(* IEC 61131-3 sources: Mizera_Tube/Plc, 88 files *)

(* ---- Aspiraz.plc ---- *)
*******************************************************************************
*   ASPIRAZ.PLC
*   ESAutomotion
*   LASER machine
*******************************************************************************
#funcdec "SetVasca.plc"

VAR
#include "Cnc.inc"

EXHAUST_MNGT:           EXHAUST;    * Vasche di aspirazione
TimeOff:                DWORD;
TON_ASP:                TON;
TON_ASPI:               TON;
TOF_ASPI:               TOF;
TON_PROGRUN:            TON;
TOF_EXEAUTO:            TOF;
appoggio:               BOOL;
END_VAR

#include "Iol.inc"
#include "Aspiraz.inc"

VAR_IN_OUT
#include "mem.inc"
END_VAR
*******************************************************************************
* Gestione Aspirazione
*******************************************************************************
FUNCTION Aspiraz

*******************************************************************************
*   Richiesta da Pulsante Aspirazione ON\OFF
*******************************************************************************

CAL  TON_PROGRUN (IN:=PRGRUN_CN0,PT:=200)
CAL  TOF_EXEAUTO (IN:=ExeAuxMode,PT:=1000)

LD   Pls_ON_OFF_Aspiratore         ** (LsGui0.31)Pulsante ON\OFF accensione Aspiratore
OR   (
LD   Pls_AspAuto                   ** (rLsGui0.11) Pulsante Abilitazione Auto Aspiratore
AND  TON_PROGRUN.Q
ANDN TOF_EXEAUTO.Q
OR (
LD   ExeAuxMode                    ** (gPlc0.29)Esecuzione ausiliaria 1000.PGM
AND  exeaux_for_mancut               ** (LsPlc47.8) manual cut request
)
)
ANDN %PlcOp0.2                     ** DryRun
ST   appoggio

LD   %Cost_User9
MUL  1000
ST   TimeOff

CAL  TON_ASPI (IN:=appoggio,PT:=100)
CAL  TOF_ASPI (IN:=TON_ASPI.Q,PT:=TimeOff)

LD   TOF_ASPI.Q
ST   O_START_ASPIRATORE            ** Command START for Aspiration system
ST   AspOnOffLED                   ** (LsPlc11.17) LED Comando ON\OFF Aspiratore

LDN  O_START_ASPIRATORE            ** Command START for Aspiration system
ST   O_STOP_ASPIRATORE             ** Command STOP for Aspiration system

***************************************
*   EXHAUST FAN
***************************************

LD   %ax27.ra3.14        * Axis referenced
AND  %ax28.ra3.14        * Axis referenced
ST   EXHAUST_MNGT.xEnab

LD   0
ST   EXHAUST_MNGT.x5axes

LD   27
ST   EXHAUST_MNGT.xNumXaxis

LD   28
ST   EXHAUST_MNGT.xNumYaxis

LD   %CostK56           * Sovrapposizione
ST   EXHAUST_MNGT.xQtaSovrap

LD   %CostK57           * Tempo apertura
ST   EXHAUST_MNGT.xTimerOff

CAL  EXHAUST_MNGT                  ** Vasche di aspirazione

***************************************

LD   EXHAUST_MNGT.yOut1.0
AND  Pls_AspAuto                   ** (rLsGui0.11) Pulsante Abilitazione Auto Aspiratore
ST   O_APERTURA_ASPIRAZIONE_1      ** Aspiraz 1
ST   %GenVasche.GV_ParDW1.0         * led for GUI

LD   EXHAUST_MNGT.yOut1.1
AND  Pls_AspAuto                   ** (rLsGui0.11) Pulsante Abilitazione Auto Aspiratore
ST   O_APERTURA_ASPIRAZIONE_2      ** Aspiraz 2
ST   %GenVasche.GV_ParDW1.1         * led for GUI

LD   EXHAUST_MNGT.yOut1.2
AND  Pls_AspAuto                   ** (rLsGui0.11) Pulsante Abilitazione Auto Aspiratore
ST   O_APERTURA_ASPIRAZIONE_3      ** Aspiraz 3
ST   %GenVasche.GV_ParDW1.2         * led for GUI

LD   EXHAUST_MNGT.yOut1.3
AND  Pls_AspAuto                   ** (rLsGui0.11) Pulsante Abilitazione Auto Aspiratore
ST   O_APERTURA_ASPIRAZIONE_4      ** Aspiraz 4
ST   %GenVasche.GV_ParDW1.3         * led for GUI

LD   EXHAUST_MNGT.yOut1.4
AND  Pls_AspAuto                   ** (rLsGui0.11) Pulsante Abilitazione Auto Aspiratore
ST   O_APERTURA_ASPIRAZIONE_5      ** Aspiraz 5
ST   %GenVasche.GV_ParDW1.4         * led for GUI

LD   EXHAUST_MNGT.yOut1.5
AND  Pls_AspAuto                   ** (rLsGui0.11) Pulsante Abilitazione Auto Aspiratore
ST   O_APERTURA_ASPIRAZIONE_6      ** Aspiraz 6
ST   %GenVasche.GV_ParDW1.5         * led for GUI

LD   EXHAUST_MNGT.yOut1.6
AND  Pls_AspAuto                   ** (rLsGui0.11) Pulsante Abilitazione Auto Aspiratore
ST   O_APERTURA_ASPIRAZIONE_7      ** Aspiraz 7
ST   %GenVasche.GV_ParDW1.6         * led for GUI

LD   EXHAUST_MNGT.yOut1.7
AND  Pls_AspAuto                   ** (rLsGui0.11) Pulsante Abilitazione Auto Aspiratore
ST   O_APERTURA_ASPIRAZIONE_8      ** Aspiraz 8
ST   %GenVasche.GV_ParDW1.7         * led for GUI

LD   EXHAUST_MNGT.yOut1.8
AND  Pls_AspAuto                   ** (rLsGui0.11) Pulsante Abilitazione Auto Aspiratore
ST   O_APERTURA_ASPIRAZIONE_9      ** Aspiraz 9
ST   %GenVasche.GV_ParDW1.8         * led for GUI

LD   EXHAUST_MNGT.yOut1.9
AND  Pls_AspAuto                   ** (rLsGui0.11) Pulsante Abilitazione Auto Aspiratore
ST   O_APERTURA_ASPIRAZIONE_10     ** Aspiraz 10
ST   %GenVasche.GV_ParDW1.9         * led for GUI

LD   EXHAUST_MNGT.yOut1.10
AND  Pls_AspAuto                   ** (rLsGui0.11) Pulsante Abilitazione Auto Aspiratore
ST   O_APERTURA_ASPIRAZIONE_11     ** Aspiraz 11
ST   %GenVasche.GV_ParDW1.10         * led for GUI

LD   EXHAUST_MNGT.yOut1.11
AND  Pls_AspAuto                   ** (rLsGui0.11) Pulsante Abilitazione Auto Aspiratore
ST   O_APERTURA_ASPIRAZIONE_12     ** Aspiraz 12
ST   %GenVasche.GV_ParDW1.11         * led for GUI

LD   EXHAUST_MNGT.yOut1.12
AND  Pls_AspAuto                   ** (rLsGui0.11) Pulsante Abilitazione Auto Aspiratore
ST   O_APERTURA_ASPIRAZIONE_13     ** Aspiraz 13
ST   %GenVasche.GV_ParDW1.12         * led for GUI

LD   EXHAUST_MNGT.yOut1.13
AND  Pls_AspAuto                   ** (rLsGui0.11) Pulsante Abilitazione Auto Aspiratore
ST   O_APERTURA_ASPIRAZIONE_14     ** Aspiraz 14
ST   %GenVasche.GV_ParDW1.13         * led for GUI

LD   EXHAUST_MNGT.yOut1.14
AND  Pls_AspAuto                   ** (rLsGui0.11) Pulsante Abilitazione Auto Aspiratore
ST   O_APERTURA_ASPIRAZIONE_15     ** Aspiraz 15
ST   %GenVasche.GV_ParDW1.14         * led for GUI

LD   EXHAUST_MNGT.yOut1.15
AND  Pls_AspAuto                   ** (rLsGui0.11) Pulsante Abilitazione Auto Aspiratore
ST   O_APERTURA_ASPIRAZIONE_16     ** Aspiraz 16
ST   %GenVasche.GV_ParDW1.15         * led for GUI

LD   EXHAUST_MNGT.yOut1.16
AND  Pls_AspAuto                   ** (rLsGui0.11) Pulsante Abilitazione Auto Aspiratore
ST   O_APERTURA_ASPIRAZIONE_17     ** Aspiraz 17
ST   %GenVasche.GV_ParDW1.16         * led for GUI

LD   EXHAUST_MNGT.yOut1.17
AND  Pls_AspAuto                   ** (rLsGui0.11) Pulsante Abilitazione Auto Aspiratore
ST   O_APERTURA_ASPIRAZIONE_18     ** Aspiraz 18
ST   %GenVasche.GV_ParDW1.17         * led for GUI

LD   EXHAUST_MNGT.yOut1.18
AND  Pls_AspAuto                   ** (rLsGui0.11) Pulsante Abilitazione Auto Aspiratore
ST   O_APERTURA_ASPIRAZIONE_19     ** Aspiraz 19
ST   %GenVasche.GV_ParDW1.18         * led for GUI

LD   EXHAUST_MNGT.yOut1.19
AND  Pls_AspAuto                   ** (rLsGui0.11) Pulsante Abilitazione Auto Aspiratore
ST   O_APERTURA_ASPIRAZIONE_20     ** Aspiraz 20
ST   %GenVasche.GV_ParDW1.19         * led for GUI

LD   EXHAUST_MNGT.yOut1.20
AND  Pls_AspAuto                   ** (rLsGui0.11) Pulsante Abilitazione Auto Aspiratore
ST   O_APERTURA_ASPIRAZIONE_21     ** Aspiraz 21
ST   %GenVasche.GV_ParDW1.20         * led for GUI

LD   EXHAUST_MNGT.yOut1.21
AND  Pls_AspAuto                   ** (rLsGui0.11) Pulsante Abilitazione Auto Aspiratore
ST   O_APERTURA_ASPIRAZIONE_22     ** Aspiraz 22
ST   %GenVasche.GV_ParDW1.21         * led for GUI

LD   EXHAUST_MNGT.yOut1.22
AND  Pls_AspAuto                   ** (rLsGui0.11) Pulsante Abilitazione Auto Aspiratore
ST   O_APERTURA_ASPIRAZIONE_23     ** Aspiraz 23
ST   %GenVasche.GV_ParDW1.22         * led for GUI

LD   EXHAUST_MNGT.yOut1.23
AND  Pls_AspAuto                   ** (rLsGui0.11) Pulsante Abilitazione Auto Aspiratore
ST   O_APERTURA_ASPIRAZIONE_24     ** Aspiraz 24
ST   %GenVasche.GV_ParDW1.23         * led for GUI

**********************************************************************
* ASPIRATORE ERROR MANAGEMENT
**********************************************************************
LD     O_START_ASPIRATORE     * (dryrun condition is included)
ANDN   I_I_ASPIRATORE_OK
ST     appoggio

CAL    TON_ASP(IN:=appoggio,PT:=1000)
LD     TON_ASP.Q
S      %PLCerr5.15

LD     Pul_Reset
R      %PLCerr5.15

*******************************************************************************
END_FUNCTION

(* ---- Barriere.plc ---- *)
*******************************************************************************
*   BARRIERE.PLC
*   ESAutomotion
*   LASER machine
*******************************************************************************
VAR
#include "Cnc.inc"

S_Carico_lam_in_esecuzione:     BOOL;   * S\Carico lamiera in esecuzione
Rit_pls_reset_barriere:         BOOL;   * Ritardo Fronte di discesa pressione Pls Reset barriere
TOF_ps_reset_barriere:          TOF;    * Ritardo pressione Pls Reset barriere
FPN_RESET_BARR:                 TRIG;   * Fronte salita\discesa pulsante Reset Barriere
END_VAR

VAR_IN_OUT
#include "mem.inc"
END_VAR

#include "Iol.inc"

******************************************************************************
*   * Gestione Barriere ottiche
******************************************************************************
FUNCTION Barriere

LD  I_I_BARRIERE_SCARICO_OK	       ** M81.31 Barriere ottiche scarico lamiera OK
ST  Barriere_ottiche_OK  		        ** M100.6  Barriere ottiche in sicurezza

***************************************
* Fronte pulsante Reset Barriere
***************************************
CAL  FPN_RESET_BARR(CLK=I_I_PLS_RESET_BARRIERE) ** Fronte salita\discesa pulsante Reset Barriere

LD   FPN_RESET_BARR.Q 		** Fronte salita\discesa pulsante Reset Barriere
AND  I_I_PLS_RESET_BARRIERE	       ** M89.26 Pulsante reset barriere
ST   FP_PS_RESET_BARRIERE		        ** M100.9  Fronte di salita pulsante Reset Barriere

LD   FPN_RESET_BARR.Q 		** Fronte salita\discesa pulsante Reset Barriere
ANDN I_I_PLS_RESET_BARRIERE	       ** M89.26 Pulsante reset barriere
ST   FN_PS_RESET_BARRIERE		        ** M100.10  Fronte di discesa pulsante Reset Barriere

***************************************
* Ritardo pressione Pulsante Reset barriere
***************************************
CAL  TOF_ps_reset_barriere(IN=FN_PS_RESET_BARRIERE,PT=500) ** Ritardo pressione Pls Reset barriere

LD   TOF_ps_reset_barriere.Q
ST   Rit_pls_reset_barriere      	 ** Ritardo Fronte di discesa pressione Pls Reset barriere

***************************************
* Allarme : BARRIERA OTTICA LATO
* PULSANTIERA INTERVENUTA CON
* SCARICO LAMIERA IN ESECUZIONE
***************************************
LD   MACCHINA_OK      		           ** M100.1  Macchina OK
AND  S_Carico_lam_in_esecuzione    ** S\Carico lamiera in esecuzione
ANDN Barriere_ottiche_OK 	         ** M100.6  Barriere ottiche in sicurezza
S    %PLCerr6.8                  	** PLC Err 200 Barriera ottica lato pulsantiera intervenuta

LD   RESET_ALLARMI 		              ** M100.4  Cancellazione allarmi attiva
OR   Rit_pls_reset_barriere      	 ** Ritardo Fronte di discesa pressione Pls Reset barriere
R    %PLCerr6.8                  	** PLC Err 200 Barriera ottica lato pulsantiera intervenuta

***************************************
* Messaggio: Ripristinare Barriera
* ottica lato pulsantiera intervenuta
***************************************
LD   MACCHINA_OK      	            ** M100.1  Macchina OK
ANDN S_Carico_lam_in_esecuzione    ** S\Carico lamiera in esecuzione
ANDN Barriere_ottiche_OK 	         ** M100.6  Barriere ottiche in sicurezza
S    %PLCmsg6.8               	** PLC Msg 200 Ripristinare barriera lato pulsant. intervenuta

LD   RESET_ALLARMI 		              ** M100.4  Cancellazione allarmi attiva
OR   Rit_pls_reset_barriere      	 ** Ritardo Fronte di discesa pressione Pls Reset barriere
OR   %PLCerr6.8                  	** PLC Err 200 Barriera ottica lato pulsantiera intervenuta
R    %PLCmsg6.8               	** PLC Msg 200 Ripristinare barriera lato pulsant. intervenuta

END_FUNCTION

(* ---- BLDFeed.plc ---- *)
#funcdec "FBAux.plc"

VAR_IN_OUT
BLDFEED_72_85_Percent    AT %UNLOADER.values44;
BLDFEED_73_86_Percent    AT %UNLOADER.values45;
BLDFEED_74_87_Percent    AT %UNLOADER.values46;
BLDFEED_75_88_Percent    AT %UNLOADER.values47;
END_VAR

VAR
BLDFEED_72_85:    CALC_BLD_FEED;
BLDFEED_73_86:    CALC_BLD_FEED;
BLDFEED_74_87:    CALC_BLD_FEED;
BLDFEED_75_88:    CALC_BLD_FEED;
END_VAR

FUNCTION BLEND_FEEDRATE

*//=============================================================================
*// Unloading Flaps On Each Support
*//=============================================================================
CAL BLDFEED_72_85(xEn:=%cn7.cc1.2 ,xH:=85 ,xV:=72 ,xVPercent:=80)
CAL BLDFEED_73_86(xEn:=%cn7.cc1.3 ,xH:=86 ,xV:=73 ,xVPercent:=80)
CAL BLDFEED_74_87(xEn:=%cn7.cc1.4 ,xH:=87 ,xV:=74 ,xVPercent:=80)
CAL BLDFEED_75_88(xEn:=%cn7.cc1.5 ,xH:=88 ,xV:=75 ,xVPercent:=80)

LD  BLDFEED_72_85.yPercent
ST  BLDFEED_72_85_Percent

LD  BLDFEED_73_86.yPercent
ST  BLDFEED_73_86_Percent

LD  BLDFEED_74_87.yPercent
ST  BLDFEED_74_87_Percent

LD  BLDFEED_75_88.yPercent
ST  BLDFEED_75_88_Percent

END_FUNCTION

(* ---- CalPipe.plc ---- *)
*******************************************************************************
*   PIPE CALIBRATION
*   ESAutomotion
*   LASER machine
* Y  G2292 X(%CalPipe.DimXPipe/1000)  Y(%CalPipe.DimYPipe/1000)   Z(%CalPipe.DimZPipe/1000)  U(%CalPipe.DimUPipe/1000)  V(%CalPipe.DimVPipe/1000) W(%CalPipe.DimWPipe/1000) J(%CalPipe.Round/1000) TYPE 1
* Y G2292 X(%CalPipe.DimXPipe1/1000)  Y(%CalPipe.DimYPipe1/1000)  Z(%CalPipe.DimZPipe1/1000) U(%CalPipe.DimUPipe1/1000) V(%CalPipe.DimVPipe1/1000)W(%CalPipe.DimWPipe1/1000)J(%CalPipe.Round1/1000) TYPE 2
* X  G2292 X(%CalPipe.DimXPipe/1000)  Y(%CalPipe.DimYPipe/1000)   Z(%CalPipe.DimZPipe/1000)  U(%CalPipe.DimUPipe/1000)  V(%CalPipe.DimVPipe/1000) W(%CalPipe.DimWPipe/1000) I(%CalPipe.Round/1000) TYPE 1
* X G2292 X(%CalPipe.DimXPipe1/1000)  Y(%CalPipe.DimYPipe1/1000)  Z(%CalPipe.DimZPipe1/1000) U(%CalPipe.DimUPipe1/1000) V(%CalPipe.DimVPipe1/1000)W(%CalPipe.DimWPipe1/1000)I(%CalPipe.Round1/1000) TYPE 2
*******************************************************************************
VAR
#include "cnc.inc"

RTRIG_CHANG_OPT1:     R_TRIG;
RTRIG_CHANG_OPT2:     R_TRIG;
RTRIG_CHANG_OPT3:     R_TRIG;
RTRIG_CHANG_OPT4:     R_TRIG;
FTRIG_PRGRUN:         F_TRIG;
R_TRIG_NO_SEL:        R_TRIG;
RTRIG_PAR_COPY:       R_TRIG;
RTRIG_RES_CAL_X:      R_TRIG;
RTRIG_RES_CAL_Y:      R_TRIG;
appoggio:               BOOL;
END_VAR

#include "iol.inc"
#include "pipe.inc"

VAR_IN_OUT
#include "mem.inc"
END_VAR

*******************************************************************************
*   Function: cancellazione tabella di calibrazione 2D e 3D
*******************************************************************************
FUNCTION RES_TAB_2D_3D

LD   3                  * Type=nutator
ST   T2D_TAB_T_KINE
ST   T3D_TAB_T_KINE

LD   0
ST   T2D_T_OART_X0
ST   T3D_T_OART_X0

LD   0
ST   T2D_T_OART_Y0
ST   T3D_T_OART_Y0

LD   0
ST   T2D_T_OART_Z0
ST   T3D_T_OART_Z0

***6 ST   T2D_T_OART_ORIENT
***6 ST   T3D_T_OART_ORIENT

LD   0
ST   T2D_T_OART_FRAME_C
ST   T3D_T_OART_FRAME_C

LD   0
ST   T2D_T_OART_FRAME_B
ST   T3D_T_OART_FRAME_B

LD   0
ST   T2D_T_OART_FRAME_A
ST   T3D_T_OART_FRAME_A

*** -90
LD   90                 * SET !
MUL  -1
MUL  1000
ST   T2D_T_OART_EC
ST   T3D_T_OART_EC

LD   0                  * SET !
ST   T2D_T_OART_ECREV
ST   T3D_T_OART_ECREV

*** 9 ST   T2D_T_OART_ECAX
*** 9 ST   T3D_T_OART_ECAX

LD   0
ST   T2D_T_OART_X1
ST   T3D_T_OART_X1

LD   0
ST   T2D_T_OART_Y1
ST   T3D_T_OART_Y1

LD   0
ST   T2D_T_OART_TILT
ST   T3D_T_OART_TILT

*** -90
LD   90                 * SET !
MUL  -1
MUL  1000
ST   T2D_T_OART_EB
ST   T3D_T_OART_EB

LD   0                  * SET !
ST   T2D_T_OART_EBREV
ST   T3D_T_OART_EBREV

LD   0
ST   T2D_T_OART_EBAX
ST   T3D_T_OART_EBAX

LD   0
ST   T2D_T_OART_X2
ST   T3D_T_OART_X2

LD   0
ST   T2D_T_OART_Y2
ST   T3D_T_OART_Y2

LD   0
ST   T2D_T_OART_Z2
ST   T3D_T_OART_Z2

LD   0
ST   T2D_T_OART_CAMBER
ST   T3D_T_OART_CAMBER

LD   0
ST   T2D_T_OART_FRAME2_C
ST   T3D_T_OART_FRAME2_C

LD   0
ST   T2D_T_OART_FRAME2_B
ST   T3D_T_OART_FRAME2_B

LD   0
ST   T2D_T_OART_FRAME2_A
ST   T3D_T_OART_FRAME2_A

END_FUNCTION

*******************************************************************************
FUNCTION PIPE_CALIBRATION

**
* Force Factory Table
LD   6
ST   %CalPipe.BackupTable                  * Factory table

* Safeties on option selections

***
CAL  RTRIG_CHANG_OPT1(CLK:=SquarePipeCal) ** (CalPipe.General.0) Table calibration for square pipe

LD   RTRIG_CHANG_OPT1.Q
JMPCN no_pipe_cal_round1
LD   ALWAYS_ONE                    ** PLCFLAGS.1  Flag sempre stato on
R    RoundPipeCal                  ** (CalPipe.General.1) Table calibration for round pipe
no_pipe_cal_round1:

CAL  RTRIG_CHANG_OPT2(CLK:=RoundPipeCal) ** (CalPipe.General.1) Table calibration for round pipe

LD   RTRIG_CHANG_OPT2.Q
JMPCN no_pipe_cal_round2
LD   ALWAYS_ONE                    ** PLCFLAGS.1  Flag sempre stato on
R    SquarePipeCal                 ** (CalPipe.General.0) Table calibration for square pipe
no_pipe_cal_round2:

* At least select one state
LDN   SquarePipeCal                ** (CalPipe.General.0) Table calibration for square pipe
ANDN  RoundPipeCal                 ** (CalPipe.General.1) Table calibration for round pipe
ST    appoggio

CAL  R_TRIG_NO_SEL (CLK:= appoggio)

LD   R_TRIG_NO_SEL.Q
JMPCN no_auto_select
LD   ALWAYS_ONE                    ** PLCFLAGS.1  Flag sempre stato on
S    SquarePipeCal                 ** (CalPipe.General.0) Table calibration for square pipe
no_auto_select:
***
* Auto Reset when pipe axis is selected

CAL  RTRIG_CHANG_OPT3(CLK:=PipeAlongX) ** (CalPipe.General.4) Pipe is cutted along X axis

LD   RTRIG_CHANG_OPT3.Q
JMPCN no_pipe_cal_x
LD   ALWAYS_ONE                    ** PLCFLAGS.1  Flag sempre stato on
R    PipeAlongY                    ** (CalPipe.General.5) Pipe is cutted along Y axis
no_pipe_cal_x:

CAL  RTRIG_CHANG_OPT4(CLK:=PipeAlongY) ** (CalPipe.General.5) Pipe is cutted along Y axis

LD   RTRIG_CHANG_OPT4.Q
JMPCN no_pipe_cal_y
LD   ALWAYS_ONE                    ** PLCFLAGS.1  Flag sempre stato on
R    PipeAlongX                    ** (CalPipe.General.4) Pipe is cutted along X axis
no_pipe_cal_y:

***
* Reset of Pipe calibration result

LD   PipeAlongX                    ** (CalPipe.General.4) Pipe is cutted along X axis
AND  ResetPipeCal                  ** (CalPipe.General.8) Button to reset the value of calibration
ST   appoggio

CAL  RTRIG_RES_CAL_X (CLK:=appoggio)

LD   PipeAlongY                    ** (CalPipe.General.5) Pipe is cutted along Y axis
AND  ResetPipeCal                  ** (CalPipe.General.8) Button to reset the value of calibration
ST   appoggio

CAL  RTRIG_RES_CAL_Y (CLK:=appoggio)

**
* Preset of table ( X or Y )

LD   RTRIG_CHANG_OPT3.Q            * Pipe is along X axis
OR   RTRIG_RES_CAL_X.Q
ANDN ON_ONE_SCAN                   ** PLCFLAGS.8  Flag on alla prima scansione PLC
JMPCN no_copy_X_par

RES_TAB_2D_3D           * Cancellazione tabella per 2D e 3D

LD   3
ST   TAB_T_KINE

LD   6
ST   T_OART_ORIENT

LD   90
MUL  -1
MUL  1000
ST   T_OART_EC

LD   9
ST   T_OART_ECAX

LD   ALWAYS_ZERO                   ** PLCFLAGS.0  Flag sempre stato off
ST   T_OART_X1
ST   T_OART_Y1
ST   T_OART_X0
ST   T_OART_Y0
ST   T_OART_Z0

LD   90
MUL  -1
MUL  1000
ST   T_OART_EB

LD   ALWAYS_ZERO                   ** PLCFLAGS.0  Flag sempre stato off
ST   T_OART_FRAME2_A
no_copy_X_par:

LD   RTRIG_CHANG_OPT4.Q           * Pipe is along Y axis
OR   RTRIG_RES_CAL_Y.Q
ANDN ON_ONE_SCAN                   ** PLCFLAGS.8  Flag on alla prima scansione PLC
JMPCN no_copy_Y_par

RES_TAB_2D_3D           * Cancellazione tabella per 2D e 3D

LD   3
ST   TAB_T_KINE

LD   8
ST   T_OART_ORIENT

LD   90
MUL  1000
ST   T_OART_EC

LD   ALWAYS_ZERO                   ** PLCFLAGS.0  Flag sempre stato off
ST   T_OART_X1
ST   T_OART_Y1
ST   T_OART_X0
ST   T_OART_Y0
ST   T_OART_Z0

LD   9
ST   T_OART_ECAX

LD   ALWAYS_ZERO                   ** PLCFLAGS.0  Flag sempre stato off
ST   T_OART_EB

LD   90
MUL  1000
ST   T_OART_FRAME2_A
no_copy_Y_par:
***

CAL  RTRIG_PAR_COPY (CLK:=FactoryParamCopy) ** (CalPipe.General.7) Factory parameters copy

LD   RTRIG_PAR_COPY.Q
JMPCN no_copy_to_factory

LD   TAB_T_KINE
ST   TAB_T_KINE_6

LD   T_OART_X0
ST   T_OART_X0_6

LD   T_OART_Y0
ST   T_OART_Y0_6

LD   T_OART_Z0
ST   T_OART_Z0_6

LD   T_OART_ORIENT
ST   T_OART_ORIENT_6

LD   T_OART_FRAME_C
ST   T_OART_FRAME_C_6

LD   T_OART_FRAME_B
ST   T_OART_FRAME_B_6

LD   T_OART_FRAME_A
ST   T_OART_FRAME_A_6

LD   T_OART_EC
ST   T_OART_EC_6

LD   T_OART_ECREV
ST   T_OART_ECREV_6

LD   T_OART_ECAX
ST   T_OART_ECAX_6

LD   T_OART_X1
ST   T_OART_X1_6

LD   T_OART_Y1
ST   T_OART_Y1_6

LD   T_OART_TILT
ST   T_OART_TILT_6

LD   T_OART_EB
ST   T_OART_EB_6

LD   T_OART_EBREV
ST   T_OART_EBREV_6

LD   T_OART_EBAX
ST   T_OART_EBAX_6

LD   T_OART_X2
ST   T_OART_X2_6

LD   T_OART_Y2
ST   T_OART_Y2_6

LD   T_OART_Z2
ST   T_OART_Z2_6

LD   T_OART_CAMBER
ST   T_OART_CAMBER_6

LD   T_OART_FRAME2_C
ST   T_OART_FRAME2_C_6

LD   T_OART_FRAME2_B
ST   T_OART_FRAME2_B_6

LD   T_OART_FRAME2_A
ST   T_OART_FRAME2_A_6
no_copy_to_factory:

**
* Datas for G2292 for the calibration

LD   PipeAlongY                    ** (CalPipe.General.5) Pipe is cutted along Y axis
JMPCN  no_gantry_Y

* Spindle
**
LD   %CalPipe.Side2               * Side 1
DIV   2
ST   %CalPipe.DimXPipe            * Shape Information X

LD   ALWAYS_ZERO                   ** PLCFLAGS.0  Flag sempre stato off
ST   %CalPipe.DimYPipe            * Shape Information Y

LD   %CalPipe.Side3               * Side2
DIV  2
MUL  -1
ST   %CalPipe.DimZPipe            * Shape Information Z

LD   %CalPipe.Side2               * Side 1
DIV  2
MUL  -1
ST   %CalPipe.DimUPipe            * Shape Information U

LD   %CalPipe.Lenght1             * Lenght of the Pipe
ST   %CalPipe.DimVPipe            * Shape Information V

LD   %CalPipe.Side3               * Side2
DIV  2
ST   %CalPipe.DimWPipe            * Shape Information W

LD   %CalPipe.RoundPar1           * Roundess from gui
ST   %CalPipe.Round               * Round of square pipe
**

* Tube
**
LD   SquarePipeCal                 ** (CalPipe.General.0) Table calibration for square pipe
JMPCN  no_square_type_2

LD   %CalPipe.Side0               * Side 1
DIV   2
ST   %CalPipe.DimXPipe1           * Shape Information X

LD   ALWAYS_ZERO                   ** PLCFLAGS.0  Flag sempre stato off
ST   %CalPipe.DimYPipe1           * Shape Information Y

LD   %CalPipe.Side1               * Side2
DIV  2
MUL  -1
ST   %CalPipe.DimZPipe1           * Shape Information Z

LD   %CalPipe.Side0               * Side 1
DIV  2
MUL  -1
ST   %CalPipe.DimUPipe1           * Shape Information U

LD   %CalPipe.Lenght0             * Lenght of the Pipe
ST   %CalPipe.DimVPipe1           * Shape Information V

LD   %CalPipe.Side1               * Side2
DIV  2
ST   %CalPipe.DimWPipe1           * Shape Information W

LD   %CalPipe.RoundPar0           * Roundess from gui
ST   %CalPipe.Round1              * Round of square pipe
no_square_type_2:
**

LD   RoundPipeCal                  ** (CalPipe.General.1) Table calibration for round pipe
JMPCN no_circle_type_2Y

LD   %CalPipe.Radius
ST   %CalPipe.DimXPipe1           * Shape Information X

LD   ALWAYS_ZERO                   ** PLCFLAGS.0  Flag sempre stato off
ST   %CalPipe.DimYPipe1           * Shape Information Y

LD   %CalPipe.Radius
MUL  -1
ST   %CalPipe.DimZPipe1           * Shape Information Z

LD   %CalPipe.Radius
MUL  -1
ST   %CalPipe.DimUPipe1           * Shape Information U

LD   %CalPipe.Lenght0             * Lenght of the Pipe
ST   %CalPipe.DimVPipe1           * Shape Information V

LD   %CalPipe.Radius
ST   %CalPipe.DimWPipe1           * Shape Information W

LD   %CalPipe.Radius
ST   %CalPipe.Round1              * Round of square pipe
no_circle_type_2Y:
**
no_gantry_Y:
***

LD   PipeAlongX                    ** (CalPipe.General.4) Pipe is cutted along X axis
JMPCN  no_gantry_X

* Spindle
**
LD   ALWAYS_ZERO                   ** PLCFLAGS.0  Flag sempre stato off
ST   %CalPipe.DimXPipe            * Shape Information X

LD   %CalPipe.Side2               * Side 1
DIV   2
MUL  -1
ST   %CalPipe.DimYPipe            * Shape Information Y

LD   %CalPipe.Side3               * Side2
DIV  2
MUL  -1
ST   %CalPipe.DimZPipe            * Shape Information Z

LD   %CalPipe.Lenght1             * Lenght of the Pipe
ST   %CalPipe.DimUPipe            * Shape Information U

LD   %CalPipe.Side2               * Side 1
DIV  2
ST   %CalPipe.DimVPipe            * Shape Information V

LD   %CalPipe.Side3               * Side2
DIV  2
ST   %CalPipe.DimWPipe            * Shape Information W

LD   %CalPipe.RoundPar1           * Roundess from gui
ST   %CalPipe.Round               * Round of square pipe
**

* Tube
**
LD   SquarePipeCal                 ** (CalPipe.General.0) Table calibration for square pipe
JMPCN  no_square_type_2X

LD   ALWAYS_ZERO                   ** PLCFLAGS.0  Flag sempre stato off
ST   %CalPipe.DimXPipe1           * Shape Information X

LD   %CalPipe.Side0               * Side 1
DIV   2
MUL  -1
ST   %CalPipe.DimYPipe1           * Shape Information Y

LD   %CalPipe.Side1               * Side2
DIV  2
MUL  -1
ST   %CalPipe.DimZPipe1           * Shape Information Z

LD   %CalPipe.Lenght0             * Lenght of the Pipe
ST   %CalPipe.DimUPipe1           * Shape Information U

LD   %CalPipe.Side0               * Side 1
DIV  2
ST   %CalPipe.DimVPipe1           * Shape Information V

LD   %CalPipe.Side1               * Side2
DIV  2
ST   %CalPipe.DimWPipe1           * Shape Information W

LD   %CalPipe.RoundPar0           * Roundess from gui
ST   %CalPipe.Round1              * Round of square pipe
no_square_type_2X:
**

LD   RoundPipeCal                  ** (CalPipe.General.1) Table calibration for round pipe
JMPCN no_circle_type_2X

LD   ALWAYS_ZERO                   ** PLCFLAGS.0  Flag sempre stato off
ST   %CalPipe.DimXPipe1           * Shape Information X

LD   %CalPipe.Radius
MUL  -1
ST   %CalPipe.DimYPipe1           * Shape Information Y

LD   %CalPipe.Radius
MUL  -1
ST   %CalPipe.DimZPipe1           * Shape Information Z

LD   %CalPipe.Lenght0             * Lenght of the Pipe
ST   %CalPipe.DimUPipe1           * Shape Information U

LD   %CalPipe.Radius
ST   %CalPipe.DimVPipe1           * Shape Information V

LD   %CalPipe.Radius
ST   %CalPipe.DimWPipe1           * Shape Information W

LD   %CalPipe.Radius
ST   %CalPipe.Round1              * Round of square pipe
no_circle_type_2X:
**
no_gantry_X:
***

***
** Calibration cycle request

LD   RunCalibration                ** (CalPipe.General.2) Run calibration from GUI
ANDN I_I_EMERGENZA                 ** Machine OK (no EMERG.)
ANDN EMER_GEN                      ** M0.10 Emergenza generale
S    ExePipeCalib                  ** (CalPipe.General.3) Exe Pipe Calibration

CAL  FTRIG_PRGRUN (CLK:=PRGRUN_CN0) ** M0.0 cn0.rc8.0  Programma in corso

LD   Pul_Reset                     ** (gPlc0.3)Reset pushbutton
OR   FTRIG_PRGRUN.Q
OR   I_I_EMERGENZA                 ** Machine OK (no EMERG.)
OR   EMER_GEN                      ** M0.10 Emergenza generale
R    ExePipeCalib                  ** (CalPipe.General.3) Exe Pipe Calibration

**
* Alarm Messages

LD   %cn3.cc1.5                   * Pipe axis configured
ANDN PipeAlongX                    ** (CalPipe.General.4) Pipe is cutted along X axis
ANDN PipeAlongY                    ** (CalPipe.General.5) Pipe is cutted along Y axis
ST   %PLCerr2.10                  * Pipe axis configured, but not define X OR Y

LD   PipeCalCycleTouch             ** (CalPipe0.General3) index to communicate in laser touch the setpoint for the calibration
EQ   0
JMPC no_check_limit

LD   %ax29.ra4                    * Z axis position [um]
LT   (
LD   %UnitWork.uxh0.a_z
SUB  %CalPipe.MaxErrTouchVert
)
ANDN CapacitiveTestRun
S    %PLCerr2.11                  * Pipe Vertical Overtravel, check Calibration data
no_check_limit:

**
* Pipe Spindle calibration

LD   SpindleCalProc                ** (CalPipe0.General2) index to comunicate to plc the spindle singfc start
JMPCN no_check_limit1

LD  %CalPipe.General.4            * pipe along X
JMPCN sim_no_x

LD   %ax28.ra4
DIV  1000
GT   (
LD   PosForSingFC                  ** (CalPipe.General1) Programmed position for singfc command inside spindle calibration
ADD  (
LD   %CalPipe.MaxErrTouchHoriz
DIV  1000
)
)
OR   (
LD   %ax28.ra4
DIV  1000
LT  (
LD   PosForSingFC                  ** (CalPipe.General1) Programmed position for singfc command inside spindle calibration
SUB  (
LD   %CalPipe.MaxErrTouchHoriz
DIV  1000
)
)
)
S    %PLCerr2.12                  *  Pipe Vertical Horizontal, check Calibration data
sim_no_x:

LD  %CalPipe.General.5            * pipe along y
JMPCN sim_no_y

LD  %ax27.ra4
DIV  1000
GT  (
LD   PosForSingFC                  ** (CalPipe.General1) Programmed position for singfc command inside spindle calibration
ADD  (
LD   %CalPipe.MaxErrTouchHoriz
DIV  1000
)
)
OR (
LD   %ax27.ra4
DIV  1000
LT  (
LD   PosForSingFC                  ** (CalPipe.General1) Programmed position for singfc command inside spindle calibration
SUB  (
LD   %CalPipe.MaxErrTouchHoriz
DIV  1000
)
)
)
S    %PLCerr2.12                  *  Pipe Vertical Horizontal, check Calibration data
sim_no_y:
no_check_limit1:

LD   Pul_Reset                     ** (gPlc0.3)Reset pushbutton
R    %PLCerr2.11                  * Pipe Vertical Overtravel, check Calibration data
R    %PLCerr2.12                  *  Pipe Vertical Horizontal, check Calibration data
**

LDN  PRGRUN_CN0                    ** M0.0 cn0.rc8.0  Programma in corso
JMPCN res_value
LD   ALWAYS_ZERO                   ** PLCFLAGS.0  Flag sempre stato off
ST   PipeCalCycleTouch             ** (CalPipe0.General3) index to communicate in laser touch the setpoint for the calibration
ST   SpindleCalProc                ** (CalPipe0.General2) index to comunicate to plc the spindle singfc start
res_value:

********************************************************************************
* Pipe cutting enable

LD   %UnitWork.gTravE
EQ   1
OR   (
LD   PipeAlongY                    ** (CalPipe.General.5) Pipe is cutted along Y axis
AND  (
 LD   %tab1.t_ttab.t_oart.t_dX
 LE   0
AND  (
 LD   %ax27.ra4
  LT   (
  LD   %ax27.pa21
  ADD  %LSRCostK9
    )
  )
 )
)
OR   (
LD   PipeAlongY                    ** (CalPipe.General.5) Pipe is cutted along Y axis
AND  (
 LD   %tab1.t_ttab.t_oart.t_dX
 GT   0
AND  (
 LD   %ax27.ra4
  GT   (
  LD   %ax27.pa22
  SUB  %LSRCostK9
    )
  )
 )
)
OR   (
LD   PipeAlongX                    ** (CalPipe.General.4) Pipe is cutted along X axis
AND  (
 LD   %tab1.t_ttab.t_oart.t_dY
 LE   0
AND  (
 LD   %ax28.ra4
  LT   (
  LD   %ax28.pa21
  ADD  %LSRCostK9
    )
  )
 )
)
OR   (
LD   PipeAlongX                    ** (CalPipe.General.4) Pipe is cutted along X axis
AND  (
 LD   %tab1.t_ttab.t_oart.t_dY
 GT   0
AND  (
 LD   %ax28.ra4
  LT   (
  LD   %ax28.pa22
  SUB  %LSRCostK9
    )
  )
 )
)
ST   O_O_PIPE_RUN                    * (QW710.10) Pipe cutting run
*********************************************************************************

END_FUNCTION

(* ---- ClampPi.plc ---- *)
*******************************************************************************
*   PIPE CALIBRATION
*   ESAutomotion
*   LASER machine
*   Support and clamp system for pipe
*******************************************************************************

VAR
#include "cnc.inc"

supp1up:        BOOL;    * memory for support 1 up
supp1down:      BOOL;    * memory for support 1 down
supp2up:        BOOL;    * memory for support 2 up
supp2down:      BOOL;    * memory for support 2 down
supp3up:        BOOL;    * memory for support 3 up
supp3down:      BOOL;    * memory for support 3 down
supp4up:        BOOL;    * memory for support 4 up
supp4down:      BOOL;    * memory for support 4 down
CLAMP_C1_OPEN_AUX:        BOOL;
CLAMP_C_OPEN_AUX:         BOOL;
CLAMP_C_CLOSE_AUX:        BOOL;

END_VAR

VAR_IN_OUT
#include "mem.inc"
END_VAR

#include "iol.inc"
#include "pipe.inc"

FUNCTION  CLAMP_SUPPORT

* If W axis is configured

LD   %cn3.cc1.5          * If W axis is configured
JMPCN no_pipe_axis

* Support 1

LD   %ax36.ra4           * Position of W axis in um
GT   %LSRCostK10         * Distance Support 1 down
OR   BSG_TAR                       ** rg1.0 Selezione modo REF (taratura)
ORN  MACC_TARATA                   ** (gPlc0.9)Assi tarati
OR   (
LD   %ax36.ra5           * W axis speed in um/s
DIV  1000                * mm/s
MUL  60                  * mm/min
GT   %LSRCostK56         * speed limit for support axes management
)
ST   supp1down                     ** memory for support 1 down

LDN  supp1down                     ** memory for support 1 down
ST   supp1up                       ** memory for support 1 up

* Support 2

LD   %ax36.ra4           * Position of W axis in um
GT   %LSRCostK11         * Distance Support 2 down
OR   BSG_TAR                       ** rg1.0 Selezione modo REF (taratura)
ORN  MACC_TARATA                   ** (gPlc0.9)Assi tarati
OR   (
LD   %ax36.ra5           * W axie speed in um/s
DIV  1000                * mm/s
MUL  60                  * mm/min
GT   %LSRCostK56         * speed limit for support axes management
)
ST   supp2down                     ** memory for support 2 down

LDN  supp2down                     ** memory for support 2 down
ST   supp2up                       ** memory for support 2 up

* Support 3

LD   %ax36.ra4           * Position of W axis in um
GT   %Cost_User30        * Distance Support 2 down
OR   BSG_TAR                       ** rg1.0 Selezione modo REF (taratura)
ORN  MACC_TARATA                   ** (gPlc0.9)Assi tarati
OR   (
LD   %ax36.ra5           * W axie speed in um/s
DIV  1000                * mm/s
MUL  60                  * mm/min
GT   %LSRCostK56         * speed limit for support axes management
)
ST   supp3down                     ** memory for support 3 down

LDN  supp3down                     ** memory for support 3 down
ST   supp3up                       ** memory for support 3 up

* Support 4

LD   %ax36.ra4           * Position of W axis in um
GT   %Cost_User29        * Distance Support 4 down
OR   BSG_TAR                       ** rg1.0 Selezione modo REF (taratura)
ORN  MACC_TARATA                   ** (gPlc0.9)Assi tarati
OR   (
LD   %ax36.ra5           * W axie speed in um/s
DIV  1000                * mm/s
MUL  60                  * mm/min
GT   %LSRCostK56         * speed limit for support axes management
)
ST   supp4down                     ** memory for support 4 down

LDN  supp4down                     ** memory for support 4 down
ST   supp4up                       ** memory for support 4 up

no_pipe_axis:

*-------------------------------------------------------------------------------
* If W axis is not configured,pipe along Y

LDN  %cn3.cc1.5          * If W axis is configured
AND  PipeAlongY                    ** (CalPipe.General.5) Pipe is cutted along Y axis
AND  %cn3.cc1.8          * If C axis is configured
JMPCN no_pipe_axis1
* Support 1

LD   %ax28.ra4           * Position of W axis in um
GT   %LSRCostK10         * Distance Support 1 down
OR   BSG_TAR                       ** rg1.0 Selezione modo REF (taratura)
ORN  MACC_TARATA                   ** (gPlc0.9)Assi tarati
OR   (
LD   %ax28.ra5           * W axie speed in um/s
DIV  1000                * mm/s
MUL  60                  * mm/min
GT   %LSRCostK56         * speed limit for support axes management
)
ST   supp1down                     ** memory for support 1 down

LDN  supp1down                     ** memory for support 1 down
ST   supp1up                       ** memory for support 1 up

* Support 2

LD   %ax28.ra4           * Position of W axis in um
GT   %LSRCostK11         * Distance Support 2 down
OR   BSG_TAR                       ** rg1.0 Selezione modo REF (taratura)
ORN  MACC_TARATA                   ** (gPlc0.9)Assi tarati
OR   (
LD   %ax28.ra5           * W axie speed in um/s
DIV  1000                * mm/s
MUL  60                  * mm/min
GT   %LSRCostK56         * speed limit for support axes management
)
ST   supp2down                     ** memory for support 2 down

LDN  supp2down                     ** memory for support 2 down
ST   supp2up                       ** memory for support 2 up

* Support 3

LD   %ax28.ra4           * Position of W axis in um
GT   %Cost_User30        * Distance Support 2 down
OR   BSG_TAR                       ** rg1.0 Selezione modo REF (taratura)
ORN  MACC_TARATA                   ** (gPlc0.9)Assi tarati
OR   (
LD   %ax28.ra5           * W axie speed in um/s
DIV  1000                * mm/s
MUL  60                  * mm/min
GT   %LSRCostK56         * speed limit for support axes management
)
ST   supp3down                     ** memory for support 3 down

LDN  supp3down                     ** memory for support 3 down
ST   supp3up                       ** memory for support 3 up

* Support 4

LD   %ax28.ra4           * Position of W axis in um
GT   %Cost_User29        * Distance Support 4 down
OR   BSG_TAR                       ** rg1.0 Selezione modo REF (taratura)
ORN  MACC_TARATA                   ** (gPlc0.9)Assi tarati
OR   (
LD   %ax28.ra5           * W axie speed in um/s
DIV  1000                * mm/s
MUL  60                  * mm/min
GT   %LSRCostK56         * speed limit for support axes management
)
ST   supp4down                     ** memory for support 4 down

LDN  supp4down                     ** memory for support 4 down
ST   supp4up                       ** memory for support 4 up
no_pipe_axis1:
*-------------------------------------------------------------------------------

* If W axis is not configured,pipe along X

LDN  %cn3.cc1.5          * If W axis is configured
AND  PipeAlongX                    ** (CalPipe.General.4) Pipe is cutted along X axis
AND  %cn3.cc1.8          * If C axis is configured
JMPCN no_pipe_axis2
* Support 1

LD   %ax27.ra4           * Position of W axis in um
GT   %LSRCostK10         * Distance Support 1 down
OR   BSG_TAR                       ** rg1.0 Selezione modo REF (taratura)
ORN  MACC_TARATA                   ** (gPlc0.9)Assi tarati
OR   (
LD   %ax27.ra5           * W axie speed in um/s
DIV  1000                * mm/s
MUL  60                  * mm/min
GT   %LSRCostK56         * speed limit for support axes management
)
ST   supp1down                     ** memory for support 1 down

LDN  supp1down                     ** memory for support 1 down
ST   supp1up                       ** memory for support 1 up

* Support 2

LD   %ax27.ra4           * Position of W axis in um
GT   %LSRCostK11         * Distance Support 2 down
OR   BSG_TAR                       ** rg1.0 Selezione modo REF (taratura)
ORN  MACC_TARATA                   ** (gPlc0.9)Assi tarati
OR   (
LD   %ax27.ra5           * W axie speed in um/s
DIV  1000                * mm/s
MUL  60                  * mm/min
GT   %LSRCostK56         * speed limit for support axes management
)
ST   supp2down                     ** memory for support 2 down

LDN  supp2down                     ** memory for support 2 down
ST   supp2up                       ** memory for support 2 up

* Support 3

LD   %ax27.ra4           * Position of W axis in um
GT   %Cost_User30        * Distance Support 2 down
OR   BSG_TAR                       ** rg1.0 Selezione modo REF (taratura)
ORN  MACC_TARATA                   ** (gPlc0.9)Assi tarati
OR   (
LD   %ax27.ra5           * W axie speed in um/s
DIV  1000                * mm/s
MUL  60                  * mm/min
GT   %LSRCostK56         * speed limit for support axes management
)
ST   supp3down                     ** memory for support 3 down

LDN  supp3down                     ** memory for support 3 down
ST   supp3up                       ** memory for support 3 up

* Support 4

LD   %ax27.ra4           * Position of W axis in um
GT   %Cost_User29        * Distance Support 4 down
OR   BSG_TAR                       ** rg1.0 Selezione modo REF (taratura)
ORN  MACC_TARATA                   ** (gPlc0.9)Assi tarati
OR   (
LD   %ax27.ra5           * W axie speed in um/s
DIV  1000                * mm/s
MUL  60                  * mm/min
GT   %LSRCostK56         * speed limit for support axes management
)
ST   supp4down                     ** memory for support 4 down

LDN  supp4down                     ** memory for support 4 down
ST   supp4up                       ** memory for support 4 up
no_pipe_axis2:
*-------------------------------------------------------------------------------

* Output

LD   supp1down                     ** memory for support 1 down
ST   O_O_SUPPORT_1_DOWN    * (QW710.7) Support 1 down

LD   supp1up                       ** memory for support 1 up
ST   O_O_SUPPORT_1_UP      * (QW710.6) Support 1 up

LD   supp2down                     ** memory for support 2 down
ST   O_O_SUPPORT_2_DOWN    * (QW710.9) Support 2 down

LD   supp2up                       ** memory for support 2 up
ST   O_O_SUPPORT_2_UP      * (QW710.8) Support 2 up

LD   supp3down                     ** memory for support 3 down
ST   O_O_SUPPORT_3_DOWN    * (QW710.9) Support 3 down

LD   supp3up                       ** memory for support 3 up
ST   O_O_SUPPORT_3_UP      * (QW710.8) Support 3 up

LD   supp4down                     ** memory for support 4 down
ST   O_O_SUPPORT_4_DOWN    * (QW710.9) Support 4 down

LD   supp4up                       ** memory for support 4 up
ST   O_O_SUPPORT_4_UP      * (QW710.8) Support 4 up

END_FUNCTION

(* ---- CopyPar.plc ---- *)
*******************************************************************************
*   ParCopy.plc
*   ESAutomotion
*   LASER machine
*   Dynamic Duty Power Frequency Management
*******************************************************************************

VAR
#include "Cnc.inc"

END_VAR

VAR_IN_OUT
#include "mem.inc"
END_VAR

#include "Iol.inc"

FUNCTION COPYPAR

* first scan parameters copy

LD   ON_ONE_SCAN                   ** PLCFLAGS.8  Flag on alla prima scansione PLC
JMPCN copy_first_scan

LD   Kp_X                          ** x axis Kp parameter
ST   XY_Kp                         ** (LsGui41) Axes position gain

LD   Jerk_X                        ** x axis Jerk parameter
ST   XY_Jerk                       ** (LsGui42) Axes jerk

LD   X_acc                         ** x axis max acceleration
ST   XY_Acc                        ** (LsGui43) axes acceleration

LD   X_dec                         ** x axis max deleration
ST   XY_Dec                        ** (LsGui44) axes deceleration

LD   Fir_1_X                       ** x axis fir 1 costant
ST   XY_TimeCostant_1              ** (LsGui45) fir 1

LD   Fir_2_X                       ** x axis fir 2 costant
ST   XY_TimeCostant_2              ** (LsGui46) fir 2

LD   Ffw_X                         ** x axis ffw
ST   XY_FFW                        ** (LsGui47) feed forward
copy_first_scan:

* User copy

LD CopyParamComm                   ** (LsGui3.0) Copy common parameter X-Y
JMPCN no_copy_param

* KP copy

LD   XY_Kp                         ** (LsGui41) Axes position gain
ST   Kp_X                          ** x axis Kp parameter
ST   Kp_Y                          ** y axis Kp parameter
ST   Kp_Gant                       ** U/V axis Kp parameter

* jerk copy

LD   XY_Jerk                       ** (LsGui42) Axes jerk
ST   Jerk_X                        ** x axis Jerk parameter
ST   Jerk_Y                        ** y axis Jerk parameter
ST   Jerk_Gant                     ** U/V axis Jerk parameter

* time costant 1 copy

LD   XY_TimeCostant_1              ** (LsGui45) fir 1
ST   Fir_1_X                       ** x axis fir 1 costant
ST   Fir_1_Y                       ** y axis fir 1 costant
ST   Fir_1_Gant                    ** U/V axis fir 1 costant

* time costant 2 copy

LD   XY_TimeCostant_2              ** (LsGui46) fir 2
ST   Fir_2_X                       ** x axis fir 2 costant
ST   Fir_2_Y                       ** y axis fir 2 costant
ST   Fir_2_Gant                    ** U/V axis fir 2 costant

* feed forward copy

LD   XY_FFW                        ** (LsGui47) feed forward
ST   Ffw_X                         ** x axis ffw
ST   Ffw_Y                         ** y axis ffw
ST   Ffw_Gant                      ** U/V axis ffw

* Acceleration copy

LD   XY_Acc                        ** (LsGui43) axes acceleration
ST   X_acc                         ** x axis max acceleration
ST   Y_acc                         ** y axis max acceleration
ST   Gant_acc                      ** U/V axis max acceleration

* Deceleration copy

LD   XY_Dec                        ** (LsGui44) axes deceleration
ST   X_dec                         ** x axis max deleration
ST   Y_dec                         ** y axis max deceleration
ST   Gant_dec                      ** U/V axis max deleration

**********************************************************************
* Copy of parameters of real on virtual axes

LD   Kp_X                          ** x axis Kp parameter
ST   %ax0.pa10            * x axis Kp parameter

LD   Kp_Y                          ** y axis Kp parameter
ST   %ax1.pa10            * y axis Kp parameter

LD   X_acc                         ** x axis max acceleration
ST   %ax0.pa1             * x axis max acceleration

LD   Y_acc                         ** y axis max acceleration
ST   %ax1.pa1             * y axis max acceleration

LD   Jerk_X                        ** x axis Jerk parameter
ST   %ax0.pa25            * x axis Jerk parameter

LD   Jerk_Y                        ** y axis Jerk parameter
ST   %ax1.pa25            * y axis Jerk parameter

LD   X_dec                         ** x axis max deleration
ST   %ax0.pa2             * x axis max deceleration

LD   Y_dec                         ** y axis max deceleration
ST   %ax1.pa2             * y axis max deceleration

no_copy_param:
**********************************************************************
* Find Kp for drive calculation

LD   3072
DIV  10
MUL  kp_Calc                       ** (LsGui48) Kp for calculation
DIV  10
MUL  100
DIV  Rpm_Calc                      ** (LsGui48) Rpm for Kp drive Calc
*DIV  10
*MUL  10
ST   KpDriveRes                    ** (LsGui50) Kp drive

END_FUNCTION

(* ---- EcatSafe.plc ---- *)
* Function to check by plc no any problem on the ecat fieldbus

VAR

#include "MainFast.inc"

END_VAR

#include "Iol.inc"

FUNCTION ECAT_SAFETY

**********************************************************************
* Wrong Working Counter (increasing) plc time must be slower than ethercat synch
* Receive Error counter
* DC error offset control

CAL  TON_ECAT_OK (IN:=EcatRun,PT:=5000) ** Actual Working Counter value
LD   TON_ECAT_OK.Q
ST   ECAT_OK

CAL  R_TRIG_WC (CLK:=TON_ECAT_OK.Q)        * at one when ethercat run

* Store the initial value of the counters

LD   R_TRIG_WC.Q
JMPCN  no_wc_store

LD   ActualWCounter                ** Actual Working Counter value
ST   firstWCounterVal              ** Wrong counter after statup of the ring

LD   ActualRxError                 ** Actual Receive error value
ST   firstRXError                  ** Initial RX error count

LD   ActualDCerror                 ** Actual DC errors
ST   firstDCerrVal                 ** DC error first value

no_wc_store:

* TP after first error on WCcounter appear wait synchTimeEthercat to check again
* the wrong wc counter value

LD   %cg27                           * reg time for ethercat synch
DIV  1000
ADD  16                              * not costant value need to be defined
ST   synchTimeEthercat             ** synch time for ethercat

CAL  TP_WCOUNT (IN:=WCerror,PT:=synchTimeEthercat) ** working counter error

LD   TP_WCOUNT.Q
JMPC wait_to_check

LD   %PLCFLAGS.0                     * PLCFLAGS.0  Flag sempre stato oFF
ST   WCerror                       ** working counter error

LD   ActualWCounter                ** Actual Working Counter value
GT   (
LD   firstWCounterVal              ** Wrong counter after statup of the ring
ADD  10000
)
AND  TON_ECAT_OK.Q
JMPCN  increase_count

LD   %PLCFLAGS.1                      * PLCFLAGS.1  Flag sempre stato on
ST   WCerror                       ** working counter error

LD   ActualWCounter                ** Actual Working Counter value
ST   firstWCounterVal              ** Wrong counter after statup of the ring

increase_count:
wait_to_check:

* Rx error

LD   TON_ECAT_OK.Q                   * at one when ethercat run
AND  (
LD   ActualRxError                 ** Actual Receive error value
NE   firstRXError                  ** Initial RX error count
)
ST   ErrorReceived                 ** Error recieved on ethercat ring

* DC error offset not stable error

LD   synchTime                     ** Measured cycle time(min,max)
SHL  16
ST   MeasuredCycleMin              ** min ethercat synch time

LD   MeasuredCycleMin              ** min ethercat synch time
SHR  16
ST   MeasuredCycleMin              ** min ethercat synch time

LD   synchTime                     ** Measured cycle time(min,max)
SHR  16
ST   MeasuredCycleMax              ** max ethercat synch time

LD   MeasuredCycleMax              ** max ethercat synch time
SUB  MeasuredCycleMin              ** min ethercat synch time
ABS
ST   DeltaSynch                    ** Delta Ethercat Synch

LD   ActualDCerror                 ** Actual DC errors
LT   (
LD   firstDCerrVal                 ** DC error first value
SUB  950                             * us
)
OR  (
LD   ActualDCerror                 ** Actual DC errors
GT   (
LD   firstDCerrVal                 ** DC error first value
ADD  950                             * us
)
)
OR   (
LD   DeltaSynch                    ** Delta Ethercat Synch
GT   950
)
AND  TON_ECAT_OK.Q
ST   ErrorDCoscillat               ** Error DC is oscillating too much

* Time to check the wrong counter error

LD   synchTimeEthercat             ** synch time for ethercat
ST   timeforAlarm                  ** time for alarm

CAL  TON_WCERROR (IN:=WCerror,PT:=timeforAlarm) ** working counter error

LD   TON_WCERROR.Q
ST   ErrorWCounter                 ** ethercat working counter is increasing
*

LD   ErrorWCounter                 ** ethercat working counter is increasing
AND  TON_ECAT_OK.Q
S    %PLCerr0.20                     * Wrong working counter increasing (ethercat error)

LD   ErrorReceived                 ** Error recieved on ethercat ring
AND  TON_ECAT_OK.Q
S    %PLCerr0.21                     * Rx error received on ethercat

* DC error commented for this moment, need to check the problem about dc offset
* during the loading of a picture for raster printing

*LD   ErrorDCoscillat                 * Error DC is oscillating too much
*AND  TON_ECAT_OK.Q
*S    %PLCerr0.22                      * DC error occurred (ethercat)

**********************************************************************
END_FUNCTION

(* ---- FastR.plc ---- *)
*******************************************************************************
*   FASTR.PLC (REAL)
*   ESAutomotion
*   LASER machine
*******************************************************************************
#funcdec "intgraph.plc"
#funcdec "DynMng.plc"

VAR
#include "MainFast.inc"
#include "Iof.inc"

BEVEL_INT:      InterpGraph;
END_VAR

VAR_IN_OUT
#include "mem.inc"
END_VAR

#include "Iol.inc"
#include "LsrGest.inc"

*******************************************************************************
FUNCTION FAST_REAL

*******************************************************************************
*   CAPACITIVE: PROCON, PRECITEC, PRECITEC LIKE (ECAT, CHC1000, EDS-C100 ...)
*******************************************************************************
LD   %config_machine26              * Capacitive Sensor (0=Precitec ,1=Lasermech,2= HighYag)
EQ   0
OR(
LD   %config_machine26              * Capacitive Sensor (0=Precitec ,1=Lasermech,2= HighYag)
EQ   6
)
JMPCN ANGFEEDBACK
     LD   I_PREC_CAPACITIVO
     ST   IA_A18_19_DIST_LINEAR
ANGFEEDBACK:

LD   %config_machine26              * Capacitive Sensor (0=Precitec ,1=Lasermech,2= HighYag)
EQ   4
JMPCN ECATFEEDBACK
     LD   I_ECAT_CAPACITIVO         * 0-10000 -> 0-%LSRCostK31 (20mm 20000)
	 MULDIV(M=AnalCapFeedback,D=10000)
     ST   IA_A18_19_DIST_LINEAR
ECATFEEDBACK:

LD   %config_machine26              * Capacitive Sensor (0=Precitec ,1=Lasermech,2= HighYag)
EQ   0
OR(
LD   %config_machine26              * Capacitive Sensor (0=Precitec ,1=Lasermech,2= HighYag)
EQ   4
)
OR(
LD   %config_machine26              * Capacitive Sensor (0=Precitec ,1=Lasermech,2= HighYag)
EQ   6
)
JMPCN NoPrecitec

LD   IA_A18_19_DIST_LINEAR          ** Capacitive sensor
ST   TempCapacitiveSensorPoints
ST   %C120                          * calibration and linearization of capacitive sensor

LD   %LSRCostK31                    ** Capacitive sensor range
DIV  10
ST   MaxVolt_x100

LD   AnalCapFeedback                * Capacitive analog resolution
ST   MaxADCPoints

JMP  HeadCom
NoPrecitec:

***************************************
*   EMPOWER 20MM
***************************************
LD   %config_machine26              * Capacitive Sensor (0=Precitec ,1=Lasermech,2= HighYag)
EQ   3
JMPCN no_em_sensor

LD   IA_Emower_cap
GE   %EmConfig.mincapval
JMPCN NORMALRNG
     LD   IA_Emower_cap
     SUB  %EmConfig.mincapval
     ST   TempCapacitiveSensorPoints
     ST   %C120
JMP  COM_RNG
NORMALRNG:
* To eliminate influence of ECAT with negative value linearization
     LD   0
     ST   TempCapacitiveSensorPoints
     ST   %C120
COM_RNG:

JMP  HeadCom
no_em_sensor:

***************************************
HeadCom:

*******************************************************************************
* Bevel Calibration and capacitive signal
*******************************************************************************
LD   %LSRPlcOp1.9                  ** Capacitive linearization from CNC
*ANDN CALIBRATION_CHECK             ** (C26.0) Calibration control in run
ANDN CAP_LINEAR_RUN                 ** (C26.2) Linearizzazione capacitivo in esecuzione
JMPCN no_calibration_bevel

LD   41                               * table 0?
ST   BEVEL_INT.xIndexFirstTable

LD   42                               * table 15?
ST   BEVEL_INT.xIndexSecondTable

LD   43                               * table 30?
ST   BEVEL_INT.xIndexThirdTable

LD   44                               * table 45?
ST   BEVEL_INT.xIndexFourthTable

LD   47                               * table for the interpolation angle distance
ST   BEVEL_INT.xIndexOutIntVal

LD   TempCapacitiveSensorPoints       * input signal
ST   BEVEL_INT.xInput

LD   bevAngleHead1_calc1
ST   BEVEL_INT.xActualAngle

CAL  BEVEL_INT                    ** for plc in simulation no external encoder head 1

LD   BEVEL_INT.yOutInterpVal
ST   TempCapacitiveSensorPoints
ST   %C120                         * calibration and linearization of capacitive sensor

no_calibration_bevel:

LD   TempCapacitiveSensorPoints
ST   %C121                         * VRTC VARIABLE

LD   TempCapacitiveSensorPoints
ST   Capacit_Anal                  ** (C102)Analogica Capacitivo

LD   Capacit_Anal                  ** (C102)Analogica Capacitivo
MUL  MaxVolt_x100
DIV  MaxADCPoints
ST   Capacit_Anal_Mm		             ** (C103)Analogica Capacitivo in mm

***LD   %UnitWork.gTravE
***EQ   1
***JMPCN no_pipe_calib

LD   TempCapacitiveSensorPoints
LT   (
LD   %LSRCostK2            * Soglia rilevamento fine materiale per APA %
MUL  AnalCapFeedback       *Capacitive analog resolution
DIV  100
)
ST   appoggio1

***no_pipe_calib:

LD   appoggio1
ST   ApaPlateSense                 ** (gPlc2.13)Sensore Rilevamento lamiera per "APA"

***************************************
*   Sicurezza
***************************************
LD   CUT_DISTANCE
DIV  10
ADD  25                            *  RANGE
ST   StandOff                      ** Valore distanza taglio in centesimi

LD   BlcAvX1_Sens_Capac            ** M74.3 Blocco avanz. asse X1 Sens. Capacitivo in contatto con la lamiera
OR   BlcAvY1_Sens_Capac            ** M74.6 Blocco avanz. asse Y Sens. Capacitivo in contatto con la lamiera
OR   Pul_Stop                      ** (gPlc0.2)Stop pushbutton
S    b_TipTouch                    ** (LsPlc47.7) TipTouch Attivo da MainFast

LDN  PRGSTOP_CN0                   ** (cn0.rc8.1)  Programma interrotto CN0
AND(
LD   V_Capacitivo                  ** Lettura tensione capacitivo (in centesimi di V)
LE   StandOff                      ** Valore distanza taglio in centesimi
)
ORN  PRGRUN_CN0                    ** M0.0 cn0.rc8.0  Programma in corso
R    b_TipTouch                    ** (LsPlc47.7) TipTouch Attivo da MainFast
****************************************************************

*******************************************************************************
* threshold detection for manual cut
*******************************************************************************
LD  %PLCFLAGS.0                ** PLCFLAGS.0  ALWAYS 0
ST  NozzleLosePlate            * (LsPlc47.13) Nozzle is far more then threshold

LD   exeaux_for_mancut         * (LsPlc47.8) manual cut request
*AND  M4001_REQ                 * (LsPlc47.14) M4001 request to enable height threshold detection
JMPCN no_check_threshold

*  value of cutting distance
LD   CUT_DISTANCE    * Distance height [um]
ADD  3200
ST   TmpHeightCheck                ** threshold for capacitive sensor

LD   %C121                     * Capacitive linearized signal (0-4095)
MUL  10
MUL  1000                       * convert in [um]
*DIV  4095                      * convert in [mm]
DIV  AnalCapFeedback       *Capacitive analog resolution convert in [mm]
GT   TmpHeightCheck                ** threshold for capacitive sensor
ST   NozzleLosePlate           * (LsPlc47.13) Nozzle is far more then threshold

no_check_threshold:

*******************************************************************************
*   TIP TOUCH condition disable
*******************************************************************************
LD   %LSRPlcOp0.12                 ** Disable TIP TOUCH during piercing
AND  PRGRUN_CN0                    ** M0.0 cn0.rc8.0  Programma in corso
AND  (
LD   PiercingInRun                 ** (LsPlc70) Piercing in run
EQ   1
)
AND (
LD   Capacit_Anal_Mm		             ** (C103)Analogica Capacitivo in mm
LT   500                        ** < 5.00 mm
)
ST   appoggio3

CAL  TON_TIPTOUCH(IN=appoggio3,PT=500) ** Tip touch ritardato di 500 msec

LD   TON_TIPTOUCH.Q             ** Tip touch ritardato di 500 msec
ST   TipTouchDisable               ** (LsPlc71.0) TipTouchDisable (ritardato)

*******************************************************************************
*   No Laser Shooting during cutting if X / V in holding
*******************************************************************************
LD    IN_M3_MODE
OR    IN_M4_MODE
AND   CMD_HOLDMOVING_CH3.4    * V
OR(
LD    IN_M2_MODE
OR    IN_M3_MODE
AND   CMD_HOLDMOVING_CH3.0    * X
)
AND(
      LD    %ax21.ra30
      EQ    0
)
AND(
      LD    SelectorApp
      EQ    4
)
AND   %cn0.rc8.0
AND   iso_LsronCutting
ST    Duty0WhenHoldSup

*******************************************************************************
END_FUNCTION

(* ---- FastS.PLC ---- *)
*******************************************************************************
*   FASTS.PLC (SIMULATION)
*   ESAutomotion
*   LASER machine
*******************************************************************************
#funcdec "intgraph.plc"
#funcdec "DynMng.plc"

VAR
#include "MainFast.inc"

BEVEL_INT:      InterpGraph;
spindleCalib:   BOOL;
new_tcp:        DWORD;
END_VAR

VAR_IN_OUT
#include "mem.inc"

END_VAR

#include "Iol.inc"
#include "LsrGest.inc"

*******************************************************************************
FUNCTION FAST_SIM

***************************************
* GAS valve simulation
***************************************
LD   OA_GAS                        ** Gas analog valve
ST   IA_Feedback_GAS_OUT           ** Gas proportional valve feedback (OUTPUT)

*LD   OA_GAS_HOERB                  ** Gas analog valve
*ST   IA_Feedb_HOERB_GAS_OUT        ** Hoerbiger gas proportional valve feedback (OUTPUT)

***************************************
* SIMULAZIONE INGRESSO CAPACITIVO
***************************************
LD   tcp_Z_head1_fast           * Z tcp measured of ch3
*SUB  %C162                      * Z tcp calculated of ch0
SUB  %ax50.ra4
MUL  (
LD   %vrtc1.VrSensorGain
DIV  1000
)
DIV  1000
ADD  %vrtc1.VrSensorOffset
ST   IA_A18_19_DIST_LINEAR

LD   IA_A18_19_DIST_LINEAR
GT   4095
*ORN  %uvHeads0.uvhCommand0.1        * NB !
JMPCN no_out_max

LD   4095
ST   IA_A18_19_DIST_LINEAR         ** Capacitive sensor
JMP  no_out_min

no_out_max:
LD   IA_A18_19_DIST_LINEAR
LT   0
JMPCN no_out_min

LD   0
ST   IA_A18_19_DIST_LINEAR         ** Capacitive sensor

no_out_min:
LD   IA_A18_19_DIST_LINEAR         ** Capacitive sensor
ST   %C120                         * calibration and linearization of capacitive sensor

*******************************************************************************
* Capacitive linearization
*******************************************************************************
*LD   Gest5Ax                        ** (gPlc0.0)Gestione MAcchina 5 assi
LD  %LSRPlcOp1.9                  ** Capacitive linearization from CNC
ANDN CALIBRATION_CHECK             ** (C26.0) Calibration control in run
ANDN CAP_LINEAR_RUN                 ** (C26.2) Linearizzazione capacitivo in esecuzione
JMPCN no_calibration_bevel

LD   41                               * table 0�
ST   BEVEL_INT.xIndexFirstTable

LD   42                               * table 15�
ST   BEVEL_INT.xIndexSecondTable

LD   43                               * table 30�
ST   BEVEL_INT.xIndexThirdTable

LD   44                               * table 45�
ST   BEVEL_INT.xIndexFourthTable

LD   47                               * table for the interpolation angle distance
ST   BEVEL_INT.xIndexOutIntVal

LD   bevAngleHead1_calc1
ST   BEVEL_INT.xActualAngle

*** TEST INTERNO (NON ABILITARE !)
LD   %User_Option0.10
JMPCN no_test_interno
LD   %gPlc99    * input signal
ST   BEVEL_INT.xInput
JMP  com_t

no_test_interno:
LD   IA_A18_19_DIST_LINEAR                            * input signal
ST   BEVEL_INT.xInput

com_t:
CAL   BEVEL_INT                    ** for plc in simulation no external encoder head 1

LD   %User_Option0.10
JMPCN no_test_interno2
LD   BEVEL_INT.yOutInterpVal
ST   %gPlc98
JMP  com_t2

no_test_interno2:
LD   BEVEL_INT.yOutInterpVal
ST   IA_A18_19_DIST_LINEAR         ** Capacitive sensor
com_t2:

no_calibration_bevel:

***************************************
LD   IA_A18_19_DIST_LINEAR         ** Capacitive sensor
ST   TempCapacitiveSensorPoints
ST   %C121
ST   %C120                            * input signal

LD   TempCapacitiveSensorPoints
ST   Capacit_Anal                  ** (C102)Analogica Capacitivo

LD   Capacit_Anal                  ** (C102)Analogica Capacitivo
MUL  %LSRCostK31                   ** Capacitive sensor range
DIV  1000
MUL  100			   ** Moltiplica per 100 per visualizzare le 2 cifre decimali
*DIV  4095
DIV  AnalCapFeedback       *Capacitive analog resolution
ST   Capacit_Anal_Mm		             ** (C103)Analogica Capacitivo in mm

***************************************
*   Sicurezza
***************************************
LD   CUT_DISTANCE
DIV  10
ADD  25                            *  RANGE
ST   StandOff                      ** Valore distanza taglio in centesimi

LD   BlcAvX1_Sens_Capac            ** M74.3 Blocco avanz. asse X1 Sens. Capacitivo in contatto con la lamiera
OR   BlcAvY1_Sens_Capac            ** M74.6 Blocco avanz. asse Y Sens. Capacitivo in contatto con la lamiera
OR   Pul_Stop                      ** (gPlc0.2)Stop pushbutton
S    b_TipTouch                    ** (LsPlc47.7) TipTouch Attivo da MainFast

LDN  PRGSTOP_CN0                   ** (cn0.rc8.1)  Programma interrotto CN0
AND(
LD   Capacit_Anal_Mm		             ** (C103)Analogica Capacitivo in mm
LE   StandOff                      ** Valore distanza taglio in centesimi
)
ORN  PRGRUN_CN0                    ** M0.0 cn0.rc8.0  Programma in corso
R    b_TipTouch                    ** (LsPlc47.7) TipTouch Attivo da MainFast
***************************************

*******************************************************************************
* threshold detection for manual cut
*******************************************************************************
LD  %PLCFLAGS.0                ** PLCFLAGS.0  ALWAYS 0
ST  NozzleLosePlate            * (LsPlc47.13) Nozzle is far more then threshold

LD   exeaux_for_mancut         * (LsPlc47.8) manual cut request
*AND  M4001_REQ                 * (LsPlc47.14) M4001 request to enable height threshold detection
JMPCN no_check_threshold

*  value of cutting distance
LD   CUT_DISTANCE    * Distance height [um]
ADD  3200
ST   TmpHeightCheck                ** threshold for capacitive sensor

LD   %C121                     * Capacitive linearized signal (0-4095)
MUL  10
MUL  1000                       * convert in [um]
*DIV  4095                      * convert in [mm]
DIV  AnalCapFeedback       *Capacitive analog resolution convert in [mm]
GT   TmpHeightCheck                ** threshold for capacitive sensor
ST   NozzleLosePlate           * (LsPlc47.13) Nozzle is far more then threshold

no_check_threshold:
*******************************************************************************
* Pipe Spindle calibration
*******************************************************************************
LD  %CalPipe.General.4               * pipe along X
JMPCN sim_no_x

LD  %ax28.ra4
GE  (
LD  %tab1.t_ttab.t_oart.t_dY
ADD  (
*LD   %CalPipe.Side2
LD   %M196
DIV  2
)
)
OR (
LD  %ax28.ra4
LE  (
LD  %tab1.t_ttab.t_oart.t_dY
SUB (
*LD   %CalPipe.Side2
LD   %M197
DIV 2
)
*MUL -1
)
)
ST  spindleCalib
sim_no_x:

LD  %CalPipe.General.5               * pipe along y
JMPCN sim_no_y

LD  %ax27.ra4
GE  (
LD  %tab1.t_ttab.t_oart.t_dX
ADD  (
LD   %CalPipe.Side2
DIV  2
)
)
OR (
LD  %ax27.ra4
LE  (
LD  %tab1.t_ttab.t_oart.t_dX
SUB (
LD   %CalPipe.Side2
DIV 2
)
*MUL -1
)
)
ST  spindleCalib
sim_no_y:

LD   %UnitWork.gTravE               * =1 pipe, =0 plane
EQ   0
JMPC no_pipe

LDN  spindleCalib
ST   ApaPlateSense                 ** (gPlc2.13)Sensore Rilevamento lamiera per "APA"

no_pipe:

END_FUNCTION

(* ---- Gas.plc ---- *)
*******************************************************************************
*   GAS.PLC
*   ESAutomotion
*   LASER machine - Cutting gas managment
*******************************************************************************

VAR
#include "Cnc.inc"
#include "RemContr.inc"

Appoggio:                  BOOL;
NoLastGasSet:              BOOL;
CloseAuxValve:             BOOL; * Close AUX valve
LaserShotCycleOn:          BOOL; * Laser shot cycle in progress
KeepCutGasEnab:            BOOL; * Keep cutting gas enable from table
KeepCutGasOxy:             BOOL; * Keep cutting oxygen enable from program
KeepCutGasNit:             BOOL; * Keep cutting nitrogen enable from program
KeepCutGasAir:             BOOL; * Keep cutting air enable from program
M550_REQ:                  BOOL; * M550: Gas blowing request
KeepSelManOxi:             BOOL; * Keep gas manual selection oxigen
KeepSelManNit:             BOOL; * Keep gas manual selection nitrogen
KeepSelManAir:             BOOL; * Keep gas manual selection air
KeepGasTestOn:             BOOL; * Keep gas test running
KeepValveTestOn:           BOOL; * Keep valve test running
GasTestButton:             BOOL; * Gas test button pressed
ValveTestButton:           BOOL; * Valve test button pressed
GasValveEnable:            BOOL; * Gas valves enable conditions
GasAuxValveEnable:         BOOL; * Gas extra valves enable conditions
PulsePurge_O2:             BOOL; * Pulse for start purge cycle on oxygen enable
PulsePurge_N2:             BOOL; * Pulse for start purge cycle on nitrogen enable
PulsePurge_AIR:            BOOL; * Pulse for start purge cycle on air enable
GasSelPgm:                 DWORD; * Gas selection in program (0-2)

RT_GAS_BTN:                R_TRIG;
#defcom RT_GAS_BTN.Q Pulse on a test gas button
RT_ON_O2:                  R_TRIG;
#defcom RT_ON_O2.Q Pulse on oxygen valve activation
RT_ON_N2:                  R_TRIG;
#defcom RT_ON_N2.Q Pulse on nitrogen valve activation
RT_ON_AIR:                 R_TRIG;
#defcom RT_ON_AIR.Q Pulse on cutting air valve activation

T_GASoff:                  TOF;
#defcom T_GASoff.Q Program run delayed for gas closing
T_Spurgo:                  TON;
#defcom T_Spurgo.Q End of purge time
T_BLOWNOLS:                TON;
#defcom T_BLOWNOLS.Q End of delay for piercing blowing

END_VAR

VAR_IN_OUT
#include "mem.inc"
END_VAR

#include "Iol.inc"

***************************************************************************************************
* Working gas valve managment
***************************************************************************************************
FUNCTION GestGas

* Program running with delay at the end

CAL  T_GASoff(IN=PRGRUN_CN0,PT=1000) ** M0.0 cn0.rc8.0  Programma in corso

LD   T_GASoff.Q                    ** Program run delayed for gas closing
ST   ProgRunForGas                 ** M107.10 Program running for gas managment

* Laser shot cycle running

LD   GasForLaserShot               ** (LsPlc11.2) Gas enable for laser shot
ST   LaserShotCycleOn              ** Laser shot cycle in progress

****************************************************************************************************
* M497:         Enable cutting gas from part program
* M496 or M498: Disable cutting gas from part program
* M480-481-482: Force cutting gas oxy/nit/air
****************************************************************************************************

LD   ch0_ValFunM                   ** %cn0.rc9 CH0 Registro Funcion M desde ISO
EQ   480
AND  ch0_StrobeM                   ** %cn0.rc8.4 CH0 Strobe Funcion M desde ISO
S    KeepCutGasOxy                 ** Keep cutting oxygen enable from program
R    KeepCutGasNit                 ** Keep cutting nitrogen enable from program
R    KeepCutGasAir                 ** Keep cutting air enable from program
R    KeepCutGasEnab                ** Keep cutting gas enable from table

LD   ch0_ValFunM                   ** %cn0.rc9 CH0 Registro Funcion M desde ISO
EQ   481
AND  ch0_StrobeM                   ** %cn0.rc8.4 CH0 Strobe Funcion M desde ISO
S    KeepCutGasNit                 ** Keep cutting nitrogen enable from program
R    KeepCutGasOxy                 ** Keep cutting oxygen enable from program
R    KeepCutGasAir                 ** Keep cutting air enable from program
R    KeepCutGasEnab                ** Keep cutting gas enable from table

LD   ch0_ValFunM                   ** %cn0.rc9 CH0 Registro Funcion M desde ISO
EQ   482
AND  ch0_StrobeM                   ** %cn0.rc8.4 CH0 Strobe Funcion M desde ISO
S    KeepCutGasAir                 ** Keep cutting air enable from program
R    KeepCutGasOxy                 ** Keep cutting oxygen enable from program
R    KeepCutGasNit                 ** Keep cutting nitrogen enable from program
R    KeepCutGasEnab                ** Keep cutting gas enable from table

LD   ch0_ValFunM                   ** %cn0.rc9 CH0 Registro Funcion M desde ISO
EQ   497
AND  ch0_StrobeM                   ** %cn0.rc8.4 CH0 Strobe Funcion M desde ISO
OR   (
LD   EnCommutValvole               ** (TstP15.1) Abilita Commutazione Valvole
ANDN AcqOrigOn                     ** (C18.7)  Acquisizione origine in corso
)
R    CloseAuxValve
S    KeepCutGasEnab                ** Keep cutting gas enable from table
R    KeepCutGasOxy                 ** Keep cutting oxygen enable from program
R    KeepCutGasNit                 ** Keep cutting nitrogen enable from program
R    KeepCutGasAir                 ** Keep cutting air enable from program

LD   ch0_ValFunM                   ** %cn0.rc9 CH0 Registro Funcion M desde ISO
EQ   496
AND  ch0_StrobeM                   ** %cn0.rc8.4 CH0 Strobe Funcion M desde ISO
S    CloseAuxValve
R    KeepCutGasOxy                 ** Keep cutting oxygen enable from program
R    KeepCutGasNit                 ** Keep cutting nitrogen enable from program
R    KeepCutGasAir                 ** Keep cutting air enable from program

LD   ch0_ValFunM                   ** %cn0.rc9 CH0 Registro Funcion M desde ISO
EQ   498
AND  ch0_StrobeM                   ** %cn0.rc8.4 CH0 Strobe Funcion M desde ISO
ORN  ProgRunForGas                 ** M107.10 Program running for gas managment
ORN  MACCHINA_OK                   ** M100.1  Macchina OK
R    CloseAuxValve
R    KeepCutGasEnab                ** Keep cutting gas enable from table
R    KeepCutGasOxy                 ** Keep cutting oxygen enable from program
R    KeepCutGasNit                 ** Keep cutting nitrogen enable from program
R    KeepCutGasAir                 ** Keep cutting air enable from program

LD   KeepCutGasOxy                 ** Keep cutting oxygen enable from program
OR   KeepCutGasNit                 ** Keep cutting nitrogen enable from program
OR   KeepCutGasAir                 ** Keep cutting air enable from program
OR   KeepCutGasEnab                ** Keep cutting gas enable from table
ST   GAS_prun                      ** M107.1 Cutting gas active from part program

LD   GAS_prun                      ** M107.1 Cutting gas active from part program
AND  ParClosePropV
AND (
LD   CloseAuxValve
AND  KeepCutGasEnab                ** Keep cutting gas enable from table
OR   PRGSTOP_CN0                   ** (cn0.rc8.1)  Programma interrotto CN0
)
OR(
LD   GAS_prun                      ** M107.1 Cutting gas active from part program
ANDN ParClosePropV
ANDN EnabExtraValve
AND (
LD   CloseAuxValve
AND  KeepCutGasEnab                ** Keep cutting gas enable from table
OR   PRGSTOP_CN0                   ** (cn0.rc8.1)  Programma interrotto CN0
)
)
ST   GAS_prun_close_propv

LDN  ProgRunForGas                 ** M107.10 Program running for gas managment
R    EnCommutValvole               ** (TstP15.1) Abilita Commutazione Valvole

****************************************************************************************************
* M550 - Gas blowing without laser beam
****************************************************************************************************

LD   ch0_ValFunM                   ** %cn0.rc9 CH0 Registro Funcion M desde ISO
EQ   550
AND  ch0_StrobeM                   ** %cn0.rc8.4 CH0 Strobe Funcion M desde ISO
ST   M550_REQ                      ** M550: Gas blowing request

CAL  T_BLOWNOLS (IN:=M550_REQ,PT:=%TabLsr0.L_SourceInt13) ** M550: Gas blowing request

LD   M550_REQ                      ** M550: Gas blowing request
ANDN T_BLOWNOLS.Q                  ** End of delay for piercing blowing
ST   WaitGasFlow                   ** (C56.0) M function iso wait

****************************************************************************************************
* Manual gas test cycle
****************************************************************************************************

LD   P_TestOxi                     ** (LsGui18.4) Gas oxigen test from valve page
OR   P_TestNit                     ** (LsGui18.5) Gas nitrogen test from valve page
OR   P_TestAir                     ** (LsGui18.3) Gas air test from valve page
OR   RemContrOxyON                 ** Xhc_Puls.14 Oxy On
OR   RemContrN2On                  ** Xhc_Puls.16 N2 on
OR   RemContrAirOn                 ** Xhc_Puls.15 Air On
OR   ButtGuiPurgeN2
OR   ButtGuiPurgeO2
OR   ButtGuiPurgeAIR
ST   GasTestButton                 ** Gas test button pressed

LD   P_ValTestAir                  ** (LsGui18.6) Valve air test from setting page
OR   P_ValTestOxy                  ** (LsGui18.7) Valve oxygen test from setting page
OR   P_ValTestNit                  ** (LsGui18.8) Valve nitrogen test from setting page
ST   ValveTestButton               ** Valve test button pressed

LD   GasTestButton                 ** Gas test button pressed
OR   ValveTestButton               ** Valve test button pressed
ST   Appoggio

CAL  RT_GAS_BTN(CLK:=Appoggio)

LD   RT_GAS_BTN.Q                  ** Pulse on a test gas button
ANDN KeepGasTestOn                 ** Keep gas test running
S    KeepGasTestOn                 ** Keep gas test running
ST   Appoggio

LD   RT_GAS_BTN.Q                  ** Pulse on a test gas button
ANDN Appoggio
OR   ProgRunForGas                 ** M107.10 Program running for gas managment
ORN  MACCHINA_OK                   ** M100.1  Macchina OK
OR   RESET_MACCHINA                ** M100.2  Reset macchina
OR   LaserShotCycleOn              ** Laser shot cycle in progress
R    KeepGasTestOn                 ** Keep gas test running

LD   ValveTestButton               ** Valve test button pressed
S    KeepValveTestOn               ** Keep valve test running

LDN  KeepGasTestOn                 ** Keep gas test running
R    KeepValveTestOn               ** Keep valve test running

LD   KeepGasTestOn                 ** Keep gas test running
ANDN KeepValveTestOn               ** Keep valve test running
OR   LaserShotCycleOn              ** Laser shot cycle in progress
ST   GAS_test                      ** M107.0 Test gas in progress for prop. valve

LD   GasTestButton                 ** Gas test button pressed
OR   LaserShotCycleOn              ** Laser shot cycle in progress
ST   PropTestRes                   ** M107.13 Proportional valve test reset from gas commands

****************************************************************************************************
* Keeps for manual cutting gas selection
****************************************************************************************************

LD   P_TestOxi                     ** (LsGui18.4) Gas oxigen test from valve page
OR   RemContrOxyON                 ** Xhc_Puls.14 Oxy On
OR   ButtGuiPurgeO2
OR   P_ValTestOxy                  ** (LsGui18.7) Valve oxygen test from setting page
S    KeepSelManOxi                 ** Keep gas manual selection oxigen
R    KeepSelManNit                 ** Keep gas manual selection nitrogen
R    KeepSelManAir                 ** Keep gas manual selection air

LD   P_TestNit                     ** (LsGui18.5) Gas nitrogen test from valve page
OR   RemContrN2On                  ** Xhc_Puls.16 N2 on
OR   ButtGuiPurgeN2
OR   P_ValTestNit                  ** (LsGui18.8) Valve nitrogen test from setting page
S    KeepSelManNit                 ** Keep gas manual selection nitrogen
R    KeepSelManOxi                 ** Keep gas manual selection oxigen
R    KeepSelManAir                 ** Keep gas manual selection air

LD   P_TestAir                     ** (LsGui18.3) Gas air test from valve page
OR   RemContrAirOn                 ** Xhc_Puls.15 Air On
OR   ButtGuiPurgeAIR
OR   P_ValTestAir                  ** (LsGui18.6) Valve air test from setting page
S    KeepSelManAir                 ** Keep gas manual selection air
R    KeepSelManOxi                 ** Keep gas manual selection oxigen
R    KeepSelManNit                 ** Keep gas manual selection nitrogen

LDN  KeepGasTestOn                 ** Keep gas test running
R    KeepSelManAir                 ** Keep gas manual selection air
R    KeepSelManOxi                 ** Keep gas manual selection oxigen
R    KeepSelManNit                 ** Keep gas manual selection nitrogen

****************************************************************************************************
* Gas valves command conditions
****************************************************************************************************

LD   %LSRPlcOp0.8                  ** Z axis in simulation (always in UP position)
AND  EnBlowDryRun                  ** (LsGui29.2) Enable gas blowing in dry run
AND  ProgRunForGas                 ** M107.10 Program running for gas managment
ST   GasEnabOnZUp                  ** M107.11 Gas enable conditions on Z up simulation

LD   %config_machine16
GT   0
AND  APAinRun                      ** (C18.31) APA in run (per gestione aria durante APA)
AND  ProgRunForGas                 ** M107.10 Program running for gas managment
ST   AirEnabForAPA                 ** M107.12 Cutting air enable for APA cycle

LD   GAS_prun                      ** M107.1 Cutting gas active from part program
OR   KeepGasTestOn                 ** Keep gas test running
OR   LaserShotCycleOn              ** Laser shot cycle in progress
OR   AirEnabForAPA                 ** M107.12 Cutting air enable for APA cycle
ANDN MACCH_IN_SIM                  ** M100.28 MACCHINA IN SIMULAZIONE
OR   GasEnabOnZUp                  ** M107.11 Gas enable conditions on Z up simulation
ANDN %PLCerr5.0                   ** PLC Err 160 Precitec - cassetto lente o protezione non presente
***ANDN PRGSTOP_CN0                   ** (cn0.rc8.1)  Programma interrotto CN0
ANDN ReqAcqOrig                    ** (gPlc13.1)Richiesta acquisizione origine
ANDN AcqOrigOn                     ** (C18.7)  Acquisizione origine in corso
***ANDN RETRACERUN                    ** M0.11 Ciclo di retrace in Run
ANDN DryRunOption                  ** Macchina in modo Dry Run
ANDN %LSRPlcOp0.22                 ** Pipe Welding function enabling
ST   Appoggio

LD   Appoggio
ANDN EnabExtraValve
ANDN PRGSTOP_CN0                   ** (cn0.rc8.1)  Programma interrotto CN0
OR (
LD   Appoggio
ANDN EnabExtraValve
AND (
LD   PRGSTOP_CN0                   ** (cn0.rc8.1)  Programma interrotto CN0
OR   KeepCutGasEnab                ** Keep cutting gas enable from table
)
AND  ParClosePropV
)
OR (
LD   Appoggio
AND  EnabExtraValve
)
ST   GasValveEnable                ** Gas valves enable conditions

LD   Appoggio
AND  EnabExtraValve
ANDN PRGSTOP_CN0                   ** (cn0.rc8.1)  Programma interrotto CN0
AND (
LDN  CloseAuxValve
OR   KeepGasTestOn                 ** Keep gas test running
)
ST   GasAuxValveEnable             ** Gas extra valves enable conditions

****************************************************************************************************
* Cutting gas valves command
****************************************************************************************************

LD  %TabLsr1.L_CutGas              	** Codice tipo Gas
ST   GasSelPgm                     ** Gas selection in program (0-2)

LD   PierceCutGasSelect            ** (LsIso31) Select piercing gas or cutting gas (0=cut gas,1=piercing gas)
JMPCN NoPiercingGas
LD   %TabLsr1.L_PierceGas            	** Codice tipo Gas
ST   GasSelPgm                     ** Gas selection in program (0-2)
NoPiercingGas:

LD   GasSelPgm                     ** Gas selection in program (0-2)
EQ   0
AND  KeepCutGasEnab                ** Keep cutting gas enable from table
OR   KeepCutGasOxy                 ** Keep cutting oxygen enable from program
ANDN AirEnabForAPA                 ** M107.12 Cutting air enable for APA cycle
AND  ProgRunForGas                 ** M107.10 Program running for gas managment
OR   (
LD   SelGasPagLaser                ** (rLsGui40) Gas selection on laser page (for shoot test)
EQ   0
AND  LaserShotCycleOn              ** Laser shot cycle in progress
)
OR   KeepSelManOxi                 ** Keep gas manual selection oxigen
AND  GasValveEnable                ** Gas valves enable conditions
ST   O_O_EV_OPEN_O2                ** Elettrovalvola apertura Ossigeno

LD   GasSelPgm                     ** Gas selection in program (0-2)
EQ   1
AND  KeepCutGasEnab                ** Keep cutting gas enable from table
OR   KeepCutGasNit                 ** Keep cutting nitrogen enable from program
ANDN AirEnabForAPA                 ** M107.12 Cutting air enable for APA cycle
AND  ProgRunForGas                 ** M107.10 Program running for gas managment
OR   (
LD   SelGasPagLaser                ** (rLsGui40) Gas selection on laser page (for shoot test)
EQ   1
AND  LaserShotCycleOn              ** Laser shot cycle in progress
)
OR   KeepSelManNit                 ** Keep gas manual selection nitrogen
AND  GasValveEnable                ** Gas valves enable conditions
ST   O_O_EV_OPEN_N2                ** Elettrovalvola apertura Azoto

LD   GasSelPgm                     ** Gas selection in program (0-2)
EQ   2
AND  KeepCutGasEnab                ** Keep cutting gas enable from table
OR   KeepCutGasAir                 ** Keep cutting air enable from program
OR   AirEnabForAPA                 ** M107.12 Cutting air enable for APA cycle
AND  ProgRunForGas                 ** M107.10 Program running for gas managment
OR   (
LD   SelGasPagLaser                ** (rLsGui40) Gas selection on laser page (for shoot test)
EQ   2
AND  LaserShotCycleOn              ** Laser shot cycle in progress
)
OR   KeepSelManAir                 ** Keep gas manual selection air
AND  GasValveEnable                ** Gas valves enable conditions
ST   O_O_EV_OPEN_ARIA              ** Elettrovalvola apertura Aria taglio

LD   O_O_EV_OPEN_O2                ** Elettrovalvola apertura Ossigeno
OR   O_O_EV_OPEN_N2                ** Elettrovalvola apertura Azoto
OR   O_O_EV_OPEN_ARIA              ** Elettrovalvola apertura Aria taglio
ST   O_O_EV_OR_ALLGAS              ** M90.15 Elettrovalvola apertura di almeno un gas

LD   O_O_EV_OR_ALLGAS              ** M90.15 Elettrovalvola apertura di almeno un gas
AND  GasAuxValveEnable             ** Gas extra valves enable conditions
ST   O_O_EV_AUX_GAS                ** Elettrovalvola ausiliaria (a valle della proporzionale)

****************************************************************************************************
* Allarme : Errore nella selezione del gas di taglio
****************************************************************************************************
LD   GasSelPgm                     ** Gas selection in program (0-2)
LT   0
OR (
LD   GasSelPgm                     ** Gas selection in program (0-2)
GT   2
)
AND  ProgRunForGas                 ** M107.10 Program running for gas managment
S    %PLCerr5.10       ** PLC Err 170 Errata selezione gas di taglio

LD   RESET_ALLARMI                 ** M100.4  Cancellazione allarmi attiva
R    %PLCerr5.10       ** PLC Err 170 Errata selezione gas di taglio

****************************************************************************************************
* Richiesto Spurgo
****************************************************************************************************
CAL  RT_ON_O2(CLK=O_O_EV_OPEN_O2)  ** Elettrovalvola apertura Ossigeno
CAL  RT_ON_N2(CLK=O_O_EV_OPEN_N2)  ** Elettrovalvola apertura Azoto
CAL  RT_ON_AIR(CLK=O_O_EV_OPEN_ARIA) ** Elettrovalvola apertura Aria taglio

LD   RT_ON_O2.Q                    ** Pulse on oxygen valve activation
AND (
LD   LastGasNit                    ** (LsPlc11.6) Keep last gas open valve nitrogen
OR   LastGasAir                    ** (LsPlc11.4) Keep last gas open valve air
OR   NoLastGasSet
)
ST   PulsePurge_O2                 ** Pulse for start purge cycle on oxygen enable

LD   RT_ON_N2.Q                    ** Pulse on nitrogen valve activation
AND (
LD   LastGasOxy                    ** (LsPlc11.5) Keep last gas open valve oxygen
OR   LastGasAir                    ** (LsPlc11.4) Keep last gas open valve air
OR   NoLastGasSet
)
ST   PulsePurge_N2                 ** Pulse for start purge cycle on nitrogen enable

LD   RT_ON_AIR.Q                   ** Pulse on cutting air valve activation
AND (
LD   LastGasOxy                    ** (LsPlc11.5) Keep last gas open valve oxygen
OR   LastGasNit                    ** (LsPlc11.6) Keep last gas open valve nitrogen
OR   NoLastGasSet
)
ST   PulsePurge_AIR                ** Pulse for start purge cycle on air enable

LD   PulsePurge_O2                 ** Pulse for start purge cycle on oxygen enable
OR   PulsePurge_N2                 ** Pulse for start purge cycle on nitrogen enable
OR   PulsePurge_AIR                ** Pulse for start purge cycle on air enable
ANDN MACCH_IN_SIM                  ** M100.28 MACCHINA IN SIMULAZIONE
S    SPURGOrun                     ** M107.2 Gas purge in progress

CAL  T_Spurgo(IN=SPURGOrun,PT=Purge_time) ** M107.2 Gas purge in progress

LD   T_Spurgo.Q                    ** End of purge time
ORN  ProgRunForGas                 ** M107.10 Program running for gas managment
R    SPURGOrun                     ** M107.2 Gas purge in progress

LD   SPURGOrun                     ** M107.2 Gas purge in progress
ST   SpurgoGas                     ** (gPlc23.0) Spurgo gas in corso
ST   %PLCmsg4.4                   * Plc Msg 132 Spurgo gas in corso

****************************************************************************************************
* Keeps for last valve open
****************************************************************************************************

LD   O_O_EV_OPEN_O2                ** Elettrovalvola apertura Ossigeno
S    LastGasOxy                    ** (LsPlc11.5) Keep last gas open valve oxygen
R    LastGasNit                    ** (LsPlc11.6) Keep last gas open valve nitrogen
R    LastGasAir                    ** (LsPlc11.4) Keep last gas open valve air

LD   O_O_EV_OPEN_N2                ** Elettrovalvola apertura Azoto
S    LastGasNit                    ** (LsPlc11.6) Keep last gas open valve nitrogen
R    LastGasOxy                    ** (LsPlc11.5) Keep last gas open valve oxygen
R    LastGasAir                    ** (LsPlc11.4) Keep last gas open valve air

LD   O_O_EV_OPEN_ARIA              ** Elettrovalvola apertura Aria taglio
S    LastGasAir                    ** (LsPlc11.4) Keep last gas open valve air
R    LastGasNit                    ** (LsPlc11.6) Keep last gas open valve nitrogen
R    LastGasOxy                    ** (LsPlc11.5) Keep last gas open valve oxygen

LD   ON_ONE_SCAN                   ** PLCFLAGS.8  Flag on alla prima scansione PLC
R    LastGasOxy                    ** (LsPlc11.5) Keep last gas open valve oxygen
R    LastGasNit                    ** (LsPlc11.6) Keep last gas open valve nitrogen
R    LastGasAir                    ** (LsPlc11.4) Keep last gas open valve air

LDN  LastGasOxy                    ** (LsPlc11.5) Keep last gas open valve oxygen
ANDN LastGasNit                    ** (LsPlc11.6) Keep last gas open valve nitrogen
ANDN LastGasAir                    ** (LsPlc11.4) Keep last gas open valve air
ST   NoLastGasSet

****************************************************************************************************
* Allarmi per bassa pressione
****************************************************************************************************
LD   GasSimulated
JMPC CONDGASSIM

LD   O_O_EV_OPEN_O2                ** Elettrovalvola apertura Ossigeno
ANDN I_I_PRESSIONE_O2              ** Pressione Ossigeno OK
S    %PLCerr5.11                  ** PLC Err 171 Bassa pressione ossigeno

LD   RESET_ALLARMI                 ** M100.4  Cancellazione allarmi attiva
R    %PLCerr5.11                  ** PLC Err 171 Bassa pressione ossigeno

LD   O_O_EV_OPEN_N2                ** Elettrovalvola apertura Azoto
ANDN I_I_PRESSIONE_N2              ** Pressione Azoto OK
S    %PLCerr5.12                  ** PLC Err 172 Bassa pressione azoto

LD   RESET_ALLARMI                 ** M100.4  Cancellazione allarmi attiva
R    %PLCerr5.12                  ** PLC Err 172 Bassa pressione azoto

LD   O_O_EV_OPEN_ARIA              ** Elettrovalvola apertura Aria taglio
ANDN I_I_PRESSIONE_ARIA            ** Pressione Aria di taglio OK
S    %PLCerr5.13                  ** PLC Err 173 Bassa pressione aria taglio

LD   RESET_ALLARMI                 ** M100.4  Cancellazione allarmi attiva
R    %PLCerr5.13                  ** PLC Err 173 Bassa pressione aria taglio
CONDGASSIM:

****************************************************************************************************
* Segnalazioni su pagina video
****************************************************************************************************

LD   O_O_EV_OPEN_O2                ** Elettrovalvola apertura Ossigeno
ST   GasYV2LED                     ** (LsPlc11.15) LED Comando Valvola Ossigeno

LD   O_O_EV_OPEN_N2                ** Elettrovalvola apertura Azoto
ST   GasYV3LED                     ** (LsPlc11.16) LED Comando Valvola Azoto

LD   O_O_EV_OPEN_ARIA              ** Elettrovalvola apertura Aria taglio
ST   GasYV0LED                     ** (LsPlc11.14) LED Comando Valvola Aria Taglio

LD   O_O_EV_AUX_GAS                ** Elettrovalvola ausiliaria (a valle della proporzionale)
ST   GasYV22LED                    ** (LsPlc11.11) LED aux valve

END_FUNCTION
